LIN {X 0,Y 374.664,Z 501.893,A -85,B 0,C 180,E1 -12895.484,E2 -12895.484} C_VEL
LIN {X 0,Y 375.928,Z 486.688,A -85,B 0,C 180,E1 -12896.337,E2 -12896.337} C_VEL
LIN {X 0,Y 376.934,Z 471.292,A -85,B 0,C 180,E1 -12896.955,E2 -12896.955} C_VEL
LIN {X 0,Y 377.639,Z 455.754,A -85,B 0,C 180,E1 -12897.35,E2 -12897.35} C_VEL
LIN {X 0,Y 380.551,Z 335.489,A -85,B 0,C 180,E1 -12899.654,E2 -12899.654} C_VEL
LIN {X 0,Y 372.146,Z 316.425,A -85,B 0,C 180,E1 -12900.818,E2 -12900.818} C_VEL
LIN {X 0,Y 363.395,Z 298.754,A -85,B 0,C 180,E1 -12902.069,E2 -12902.069} C_VEL
LIN {X 0,Y 361.869,Z 293.041,A -85,B 0,C 180,E1 -12903.644,E2 -12903.644} C_VEL
LIN {X 0,Y 361.861,Z 293.034,A -85,B 0,C 180,E1 -12907.222,E2 -12907.222} C_VEL
LIN {X 0,Y 361.831,Z 293.031,A -85,B 0,C 180,E1 -12910.754,E2 -12910.754} C_VEL
LIN {X 0,Y 361.812,Z 293.041,A -85,B 0,C 180,E1 -12914.368,E2 -12914.368} C_VEL
LIN {X 0,Y 361.83,Z 293.025,A -85,B 0,C 180,E1 -12917.567,E2 -12917.567} C_VEL
LIN {X 0,Y 361.86,Z 293.038,A -85,B 0,C 180,E1 -12920.973,E2 -12920.973} C_VEL
LIN {X 0,Y 361.863,Z 293.025,A -85,B 0,C 180,E1 -12924.655,E2 -12924.655} C_VEL
LIN {X 0,Y 361.83,Z 293.023,A -85,B 0,C 180,E1 -12928.37,E2 -12928.37} C_VEL
LIN {X 0,Y 361.879,Z 293.031,A -85,B 0,C 180,E1 -12932.218,E2 -12932.218} C_VEL
LIN {X 0,Y 361.898,Z 293.029,A -85,B 0,C 180,E1 -12935.932,E2 -12935.932} C_VEL
LIN {X 0,Y 361.874,Z 293.033,A -85,B 0,C 180,E1 -12939.538,E2 -12939.538} C_VEL
LIN {X 0,Y 361.919,Z 293.024,A -85,B 0,C 180,E1 -12943.065,E2 -12943.065} C_VEL
LIN {X 0,Y 361.989,Z 293.013,A -85,B 0,C 180,E1 -12946.527,E2 -12946.527} C_VEL
LIN {X 0,Y 361.989,Z 293.016,A -85,B 0,C 180,E1 -12949.937,E2 -12949.937} C_VEL
LIN {X 0,Y 362.131,Z 293.001,A -85,B 0,C 180,E1 -12953.313,E2 -12953.313} C_VEL
LIN {X 0,Y 362.26,Z 292.984,A -85,B 0,C 180,E1 -12957.776,E2 -12957.776} C_VEL
LIN {X 0,Y 362.37,Z 292.964,A -85,B 0,C 180,E1 -12960,E2 -12960} C_VEL
LIN {X 0,Y 362.254,Z 292.985,A -85,B 0,C 180,E1 -12962.224,E2 -12962.224} C_VEL
LIN {X 0,Y 362.129,Z 293.005,A -85,B 0,C 180,E1 -12966.687,E2 -12966.687} C_VEL
LIN {X 0,Y 361.986,Z 293.014,A -85,B 0,C 180,E1 -12970.063,E2 -12970.063} C_VEL
LIN {X 0,Y 361.988,Z 293.011,A -85,B 0,C 180,E1 -12973.899,E2 -12973.899} C_VEL
LIN {X 0,Y 361.917,Z 293.024,A -85,B 0,C 180,E1 -12976.935,E2 -12976.935} C_VEL
LIN {X 0,Y 361.874,Z 293.035,A -85,B 0,C 180,E1 -12980.462,E2 -12980.462} C_VEL
LIN {X 0,Y 361.852,Z 293.04,A -85,B 0,C 180,E1 -12984.102,E2 -12984.102} C_VEL
LIN {X 0,Y 361.834,Z 293.039,A -85,B 0,C 180,E1 -12987.785,E2 -12987.785} C_VEL
LIN {X 0,Y 361.839,Z 293.037,A -85,B 0,C 180,E1 -12991.286,E2 -12991.286} C_VEL
LIN {X 0,Y 361.842,Z 293.037,A -85,B 0,C 180,E1 -12994.282,E2 -12994.282} C_VEL
LIN {X 0,Y 361.849,Z 293.034,A -85,B 0,C 180,E1 -12997.222,E2 -12997.222} C_VEL
LIN {X 0,Y 361.805,Z 293.021,A -85,B 0,C 180,E1 -13000.752,E2 -13000.752} C_VEL
LIN {X 0,Y 361.807,Z 293.04,A -85,B 0,C 180,E1 -13004.37,E2 -13004.37} C_VEL
LIN {X 0,Y 361.816,Z 293.042,A -85,B 0,C 180,E1 -13007.571,E2 -13007.571} C_VEL
LIN {X 0,Y 361.837,Z 293.035,A -85,B 0,C 180,E1 -13011.573,E2 -13011.573} C_VEL
LIN {X 0,Y 361.874,Z 293.078,A -85,B 0,C 180,E1 -13012.878,E2 -13012.878} C_VEL
LIN {X 0,Y 365.461,Z 306.162,A -85,B 0,C 180,E1 -13016.105,E2 -13016.105} C_VEL
LIN {X 0,Y 367.967,Z 316.314,A -85,B 0,C 180,E1 -13018.431,E2 -13018.431} C_VEL
LIN {X 0,Y 375.127,Z 332.742,A -85,B 0,C 180,E1 -13019.453,E2 -13019.453} C_VEL
LIN {X 0,Y 380.024,Z 358.744,A -85,B 0,C 180,E1 -13020.439,E2 -13020.439} C_VEL
LIN {X 0,Y 377.691,Z 458.455,A -85,B 0,C 180,E1 -13022.353,E2 -13022.353} C_VEL
LIN {X 0,Y 376.872,Z 484.598,A -85,B 0,C 180,E1 -13022.89,E2 -13022.89} C_VEL
LIN {X 0,Y 375.857,Z 500.037,A -85,B 0,C 180,E1 -13023.411,E2 -13023.411} C_VEL
LIN {X 0,Y 374.562,Z 514.958,A -85,B 0,C 180,E1 -13024.137,E2 -13024.137} C_VEL
LIN {X 0,Y 373.104,Z 528.815,A -85,B 0,C 180,E1 -13025.025,E2 -13025.025} C_VEL
LIN {X 0,Y 371.347,Z 542.584,A -85,B 0,C 180,E1 -13026.139,E2 -13026.139} C_VEL
LIN {X 0,Y 369.455,Z 556.024,A -85,B 0,C 180,E1 -13027.492,E2 -13027.492} C_VEL
LIN {X 0,Y 367.597,Z 568.269,A -85,B 0,C 180,E1 -13028.994,E2 -13028.994} C_VEL
LIN {X 0,Y 365.948,Z 579.825,A -85,B 0,C 180,E1 -13030.719,E2 -13030.719} C_VEL
LIN {X 0,Y 364.213,Z 590.313,A -85,B 0,C 180,E1 -13032.597,E2 -13032.597} C_VEL
LIN {X 0,Y 362.902,Z 599.362,A -85,B 0,C 180,E1 -13034.557,E2 -13034.557} C_VEL
LIN {X 0,Y 361.936,Z 606.874,A -85,B 0,C 180,E1 -13036.526,E2 -13036.526} C_VEL
LIN {X 0,Y 361.142,Z 613.884,A -85,B 0,C 180,E1 -13038.779,E2 -13038.779} C_VEL
LIN {X 0,Y 360.644,Z 619.4,A -85,B 0,C 180,E1 -13041.031,E2 -13041.031} C_VEL
LIN {X 0,Y 360.386,Z 623.572,A -85,B 0,C 180,E1 -13043.281,E2 -13043.281} C_VEL
LIN {X 0,Y 360.309,Z 626.5,A -85,B 0,C 180,E1 -13045.525,E2 -13045.525} C_VEL
LIN {X 0,Y 360.256,Z 628.244,A -85,B 0,C 180,E1 -13047.764,E2 -13047.764} C_VEL
LIN {X 0,Y 360.357,Z 628.844,A -85,B 0,C 180,E1 -13050,E2 -13050} C_VEL
LIN {X 0,Y 360.256,Z 628.237,A -85,B 0,C 180,E1 -13052.236,E2 -13052.236} C_VEL
LIN {X 0,Y 360.303,Z 626.484,A -85,B 0,C 180,E1 -13054.475,E2 -13054.475} C_VEL
LIN {X 0,Y 360.385,Z 623.553,A -85,B 0,C 180,E1 -13056.719,E2 -13056.719} C_VEL
LIN {X 0,Y 360.633,Z 619.38,A -85,B 0,C 180,E1 -13058.969,E2 -13058.969} C_VEL
LIN {X 0,Y 361.141,Z 613.854,A -85,B 0,C 180,E1 -13061.221,E2 -13061.221} C_VEL
LIN {X 0,Y 361.912,Z 606.826,A -85,B 0,C 180,E1 -13063.475,E2 -13063.475} C_VEL
LIN {X 0,Y 363.101,Z 598.089,A -85,B 0,C 180,E1 -13065.722,E2 -13065.722} C_VEL
LIN {X 0,Y 364.432,Z 588.811,A -85,B 0,C 180,E1 -13067.682,E2 -13067.682} C_VEL
LIN {X 0,Y 365.958,Z 579.723,A -85,B 0,C 180,E1 -13069.287,E2 -13069.287} C_VEL
LIN {X 0,Y 367.626,Z 568.19,A -85,B 0,C 180,E1 -13071.004,E2 -13071.004} C_VEL
LIN {X 0,Y 369.477,Z 555.931,A -85,B 0,C 180,E1 -13072.507,E2 -13072.507} C_VEL
LIN {X 0,Y 371.354,Z 542.454,A -85,B 0,C 180,E1 -13073.861,E2 -13073.861} C_VEL
LIN {X 0,Y 373.094,Z 528.68,A -85,B 0,C 180,E1 -13074.973,E2 -13074.973} C_VEL
LIN {X 0,Y 374.602,Z 514.187,A -85,B 0,C 180,E1 -13075.898,E2 -13075.898} C_VEL
LIN {X 0,Y 375.971,Z 498.225,A -85,B 0,C 180,E1 -13076.655,E2 -13076.655} C_VEL
LIN {X 0,Y 376.879,Z 483.026,A -85,B 0,C 180,E1 -13077.147,E2 -13077.147} C_VEL
LIN {X 0,Y 379.232,Z 393.182,A -85,B 0,C 180,E1 -13078.883,E2 -13078.883} C_VEL
LIN {X 0,Y 379.96,Z 358.776,A -85,B 0,C 180,E1 -13079.551,E2 -13079.551} C_VEL
LIN {X 0,Y 374.924,Z 332.033,A -85,B 0,C 180,E1 -13080.564,E2 -13080.564} C_VEL
LIN {X 0,Y 367.914,Z 315.979,A -85,B 0,C 180,E1 -13081.585,E2 -13081.585} C_VEL
LIN {X 0,Y 364.205,Z 301.343,A -85,B 0,C 180,E1 -13085.034,E2 -13085.034} C_VEL
LIN {X 0,Y 361.866,Z 293.036,A -85,B 0,C 180,E1 -13087.123,E2 -13087.123} C_VEL
LIN {X 0,Y 361.806,Z 293.044,A -85,B 0,C 180,E1 -13090.75,E2 -13090.75} C_VEL
LIN {X 0,Y 361.808,Z 293.044,A -85,B 0,C 180,E1 -13094.368,E2 -13094.368} C_VEL
LIN {X 0,Y 361.823,Z 293.039,A -85,B 0,C 180,E1 -13097.569,E2 -13097.569} C_VEL
LIN {X 0,Y 361.834,Z 293.037,A -85,B 0,C 180,E1 -13101.571,E2 -13101.571} C_VEL
LIN {X 0,Y 361.861,Z 293.031,A -85,B 0,C 180,E1 -13104.656,E2 -13104.656} C_VEL
LIN {X 0,Y 361.829,Z 293.038,A -85,B 0,C 180,E1 -13108.37,E2 -13108.37} C_VEL
LIN {X 0,Y 361.857,Z 293.033,A -85,B 0,C 180,E1 -13110.952,E2 -13110.952} C_VEL
LIN {X 0,Y 361.851,Z 293.035,A -85,B 0,C 180,E1 -13114.704,E2 -13114.704} C_VEL
LIN {X 0,Y 361.85,Z 293.033,A -85,B 0,C 180,E1 -13118.345,E2 -13118.345} C_VEL
LIN {X 0,Y 361.91,Z 293.011,A -85,B 0,C 180,E1 -13122.085,E2 -13122.085} C_VEL
LIN {X 0,Y 361.951,Z 293.024,A -85,B 0,C 180,E1 -13125.379,E2 -13125.379} C_VEL
LIN {X 0,Y 361.95,Z 292.993,A -85,B 0,C 180,E1 -13128.804,E2 -13128.804} C_VEL
LIN {X 0,Y 362.068,Z 293.008,A -85,B 0,C 180,E1 -13132.191,E2 -13132.191} C_VEL
LIN {X 0,Y 362.087,Z 292.997,A -85,B 0,C 180,E1 -13134.431,E2 -13134.431} C_VEL
LIN {X 0,Y 362.253,Z 292.98,A -85,B 0,C 180,E1 -13137.776,E2 -13137.776} C_VEL
LIN {X 0,Y 362.258,Z 292.978,A -85,B 0,C 180,E1 -13142.224,E2 -13142.224} C_VEL
LIN {X 0,Y 362.13,Z 292.996,A -85,B 0,C 180,E1 -13146.687,E2 -13146.687} C_VEL
LIN {X 0,Y 361.988,Z 293.014,A -85,B 0,C 180,E1 -13150.063,E2 -13150.063} C_VEL
LIN {X 0,Y 361.988,Z 293.015,A -85,B 0,C 180,E1 -13153.899,E2 -13153.899} C_VEL
LIN {X 0,Y 361.918,Z 293.029,A -85,B 0,C 180,E1 -13156.935,E2 -13156.935} C_VEL
LIN {X 0,Y 361.874,Z 293.008,A -85,B 0,C 180,E1 -13160.462,E2 -13160.462} C_VEL
LIN {X 0,Y 361.885,Z 293.03,A -85,B 0,C 180,E1 -13164.113,E2 -13164.113} C_VEL
LIN {X 0,Y 361.88,Z 293.013,A -85,B 0,C 180,E1 -13167.782,E2 -13167.782} C_VEL
LIN {X 0,Y 361.839,Z 293.035,A -85,B 0,C 180,E1 -13171.286,E2 -13171.286} C_VEL
LIN {X 0,Y 361.843,Z 293.036,A -85,B 0,C 180,E1 -13174.282,E2 -13174.282} C_VEL
LIN {X 0,Y 361.854,Z 293.032,A -85,B 0,C 180,E1 -13177.223,E2 -13177.223} C_VEL
LIN {X 0,Y 361.829,Z 293.037,A -85,B 0,C 180,E1 -13180.756,E2 -13180.756} C_VEL
LIN {X 0,Y 361.812,Z 293.041,A -85,B 0,C 180,E1 -13184.369,E2 -13184.369} C_VEL
LIN {X 0,Y 361.832,Z 293.039,A -85,B 0,C 180,E1 -13187.569,E2 -13187.569} C_VEL
LIN {X 0,Y 361.866,Z 293.026,A -85,B 0,C 180,E1 -13190.974,E2 -13190.974} C_VEL
LIN {X 0,Y 361.871,Z 293.028,A -85,B 0,C 180,E1 -13194.656,E2 -13194.656} C_VEL
LIN {X 0,Y 361.871,Z 293.2,A -85,B 0,C 180,E1 -13196.547,E2 -13196.547} C_VEL
LIN {X 0,Y 363.492,Z 299.001,A -85,B 0,C 180,E1 -13198.071,E2 -13198.071} C_VEL
LIN {X 0,Y 374.141,Z 320.751,A -85,B 0,C 180,E1 -13199.567,E2 -13199.567} C_VEL
LIN {X 0,Y 380.491,Z 335.431,A -85,B 0,C 180,E1 -13200.445,E2 -13200.445} C_VEL
LIN {X 0,Y 378.084,Z 434.705,A -85,B 0,C 180,E1 -13202.347,E2 -13202.347} C_VEL
LIN {X 0,Y 377.196,Z 464.75,A -85,B 0,C 180,E1 -13202.952,E2 -13202.952} C_VEL
LIN {X 0,Y 376.39,Z 480.281,A -85,B 0,C 180,E1 -13203.484,E2 -13203.484} C_VEL
LIN {X 0,Y 375.345,Z 494.194,A -85,B 0,C 180,E1 -13204.156,E2 -13204.156} C_VEL
LIN {X 0,Y 374.115,Z 507.436,A -85,B 0,C 180,E1 -13204.997,E2 -13204.997} C_VEL
LIN {X 0,Y 372.454,Z 521.009,A -85,B 0,C 180,E1 -13206.066,E2 -13206.066} C_VEL
LIN {X 0,Y 370.69,Z 534.773,A -85,B 0,C 180,E1 -13207.424,E2 -13207.424} C_VEL
LIN {X 0,Y 368.995,Z 546.126,A -85,B 0,C 180,E1 -13208.785,E2 -13208.785} C_VEL
LIN {X 0,Y 367.249,Z 557.582,A -85,B 0,C 180,E1 -13210.434,E2 -13210.434} C_VEL
LIN {X 0,Y 365.692,Z 567.22,A -85,B 0,C 180,E1 -13212.092,E2 -13212.092} C_VEL
LIN {X 0,Y 364.187,Z 576.663,A -85,B 0,C 180,E1 -13214.039,E2 -13214.039} C_VEL
LIN {X 0,Y 363.002,Z 584.521,A -85,B 0,C 180,E1 -13215.995,E2 -13215.995} C_VEL
LIN {X 0,Y 362.214,Z 590.183,A -85,B 0,C 180,E1 -13217.677,E2 -13217.677} C_VEL
LIN {X 0,Y 361.42,Z 596.35,A -85,B 0,C 180,E1 -13219.921,E2 -13219.921} C_VEL
LIN {X 0,Y 360.905,Z 601.111,A -85,B 0,C 180,E1 -13222.166,E2 -13222.166} C_VEL
LIN {X 0,Y 360.586,Z 604.598,A -85,B 0,C 180,E1 -13224.408,E2 -13224.408} C_VEL
LIN {X 0,Y 360.374,Z 606.904,A -85,B 0,C 180,E1 -13226.646,E2 -13226.646} C_VEL
LIN {X 0,Y 360.348,Z 608.08,A -85,B 0,C 180,E1 -13228.883,E2 -13228.883} C_VEL
LIN {X 0,Y 360.348,Z 608.095,A -85,B 0,C 180,E1 -13231.118,E2 -13231.118} C_VEL
LIN {X 0,Y 360.369,Z 606.98,A -85,B 0,C 180,E1 -13233.354,E2 -13233.354} C_VEL
LIN {X 0,Y 360.57,Z 604.732,A -85,B 0,C 180,E1 -13235.593,E2 -13235.593} C_VEL
LIN {X 0,Y 360.872,Z 601.3,A -85,B 0,C 180,E1 -13237.835,E2 -13237.835} C_VEL
LIN {X 0,Y 361.385,Z 596.6,A -85,B 0,C 180,E1 -13240.08,E2 -13240.08} C_VEL
LIN {X 0,Y 362.244,Z 590.194,A -85,B 0,C 180,E1 -13242.421,E2 -13242.421} C_VEL
LIN {X 0,Y 363.065,Z 583.887,A -85,B 0,C 180,E1 -13244.288,E2 -13244.288} C_VEL
LIN {X 0,Y 364.319,Z 575.879,A -85,B 0,C 180,E1 -13246.243,E2 -13246.243} C_VEL
LIN {X 0,Y 364.568,Z 574.52,A -85,B 0,C 180,E1 -13246.547,E2 -13246.547} C_VEL
LIN {X 0,Y 364.5,Z 571.102,A -85,B 0,C 180,E1 -13247.293,E2 -13247.293} C_VEL
LIN {X 0,Y 362.703,Z 565.43,A -85,B 0,C 180,E1 -13248.538,E2 -13248.538} C_VEL
LIN {X 0,Y 360.981,Z 559.353,A -85,B 0,C 180,E1 -13249.758,E2 -13249.758} C_VEL
LIN {X 0,Y 361.007,Z 555.28,A -85,B 0,C 180,E1 -13250.443,E2 -13250.443} C_VEL
LIN {X 0,Y 362.764,Z 543.878,A -85,B 0,C 180,E1 -13252.046,E2 -13252.046} C_VEL
LIN {X 0,Y 364.597,Z 532.01,A -85,B 0,C 180,E1 -13253.426,E2 -13253.426} C_VEL
LIN {X 0,Y 366.32,Z 519.162,A -85,B 0,C 180,E1 -13254.662,E2 -13254.662} C_VEL
LIN {X 0,Y 367.952,Z 505.063,A -85,B 0,C 180,E1 -13255.755,E2 -13255.755} C_VEL
LIN {X 0,Y 369.36,Z 489.844,A -85,B 0,C 180,E1 -13256.669,E2 -13256.669} C_VEL
LIN {X 0,Y 370.399,Z 475.161,A -85,B 0,C 180,E1 -13257.318,E2 -13257.318} C_VEL
LIN {X 0,Y 371.184,Z 460.482,A -85,B 0,C 180,E1 -13257.752,E2 -13257.752} C_VEL
LIN {X 0,Y 374.403,Z 337.801,A -85,B 0,C 180,E1 -13260.144,E2 -13260.144} C_VEL
LIN {X 0,Y 368.077,Z 323.029,A -85,B 0,C 180,E1 -13261.052,E2 -13261.052} C_VEL
LIN {X 0,Y 359.045,Z 304.685,A -85,B 0,C 180,E1 -13262.355,E2 -13262.355} C_VEL
LIN {X 0,Y 356.106,Z 298.924,A -85,B 0,C 180,E1 -13262.823,E2 -13262.823} C_VEL
LIN {X 0,Y 354.807,Z 293.915,A -85,B 0,C 180,E1 -13264.239,E2 -13264.239} C_VEL
LIN {X 0,Y 354.803,Z 293.915,A -85,B 0,C 180,E1 -13267.882,E2 -13267.882} C_VEL
LIN {X 0,Y 354.784,Z 293.912,A -85,B 0,C 180,E1 -13271.171,E2 -13271.171} C_VEL
LIN {X 0,Y 354.758,Z 293.92,A -85,B 0,C 180,E1 -13274.505,E2 -13274.505} C_VEL
LIN {X 0,Y 354.788,Z 293.901,A -85,B 0,C 180,E1 -13277.662,E2 -13277.662} C_VEL
LIN {X 0,Y 354.81,Z 293.913,A -85,B 0,C 180,E1 -13280.665,E2 -13280.665} C_VEL
LIN {X 0,Y 354.812,Z 293.901,A -85,B 0,C 180,E1 -13284.301,E2 -13284.301} C_VEL
LIN {X 0,Y 354.779,Z 293.908,A -85,B 0,C 180,E1 -13287.666,E2 -13287.666} C_VEL
LIN {X 0,Y 354.813,Z 293.912,A -85,B 0,C 180,E1 -13291.616,E2 -13291.616} C_VEL
LIN {X 0,Y 354.866,Z 293.901,A -85,B 0,C 180,E1 -13294.17,E2 -13294.17} C_VEL
LIN {X 0,Y 354.799,Z 293.908,A -85,B 0,C 180,E1 -13297.892,E2 -13297.892} C_VEL
LIN {X 0,Y 354.842,Z 293.903,A -85,B 0,C 180,E1 -13301.525,E2 -13301.525} C_VEL
LIN {X 0,Y 354.909,Z 293.899,A -85,B 0,C 180,E1 -13305.082,E2 -13305.082} C_VEL
LIN {X 0,Y 354.922,Z 293.9,A -85,B 0,C 180,E1 -13308.579,E2 -13308.579} C_VEL
LIN {X 0,Y 355.052,Z 293.878,A -85,B 0,C 180,E1 -13312.035,E2 -13312.035} C_VEL
LIN {X 0,Y 355.066,Z 293.882,A -85,B 0,C 180,E1 -13314.32,E2 -13314.32} C_VEL
LIN {X 0,Y 355.222,Z 293.86,A -85,B 0,C 180,E1 -13317.732,E2 -13317.732} C_VEL
LIN {X 0,Y 355.321,Z 293.841,A -85,B 0,C 180,E1 -13320,E2 -13320} C_VEL
LIN {X 0,Y 355.217,Z 293.862,A -85,B 0,C 180,E1 -13322.268,E2 -13322.268} C_VEL
LIN {X 0,Y 355.094,Z 293.88,A -85,B 0,C 180,E1 -13326.82,E2 -13326.82} C_VEL
LIN {X 0,Y 354.943,Z 293.893,A -85,B 0,C 180,E1 -13330.265,E2 -13330.265} C_VEL
LIN {X 0,Y 354.933,Z 293.891,A -85,B 0,C 180,E1 -13334.018,E2 -13334.018} C_VEL
LIN {X 0,Y 354.88,Z 293.899,A -85,B 0,C 180,E1 -13338.092,E2 -13338.092} C_VEL
LIN {X 0,Y 354.797,Z 293.91,A -85,B 0,C 180,E1 -13342.108,E2 -13342.108} C_VEL
LIN {X 0,Y 354.797,Z 293.91,A -85,B 0,C 180,E1 -13345.835,E2 -13345.835} C_VEL
LIN {X 0,Y 354.788,Z 293.916,A -85,B 0,C 180,E1 -13349.684,E2 -13349.684} C_VEL
LIN {X 0,Y 354.778,Z 293.913,A -85,B 0,C 180,E1 -13352.334,E2 -13352.334} C_VEL
LIN {X 0,Y 354.81,Z 293.912,A -85,B 0,C 180,E1 -13355.699,E2 -13355.699} C_VEL
LIN {X 0,Y 354.761,Z 293.908,A -85,B 0,C 180,E1 -13359.413,E2 -13359.413} C_VEL
LIN {X 0,Y 354.778,Z 293.917,A -85,B 0,C 180,E1 -13362.867,E2 -13362.867} C_VEL
LIN {X 0,Y 354.756,Z 293.918,A -85,B 0,C 180,E1 -13366.103,E2 -13366.103} C_VEL
LIN {X 0,Y 354.757,Z 293.919,A -85,B 0,C 180,E1 -13369.176,E2 -13369.176} C_VEL
LIN {X 0,Y 354.813,Z 293.951,A -85,B 0,C 180,E1 -13372.264,E2 -13372.264} C_VEL
LIN {X 0,Y 358.306,Z 306.545,A -85,B 0,C 180,E1 -13375.468,E2 -13375.468} C_VEL
LIN {X 0,Y 360.733,Z 316.15,A -85,B 0,C 180,E1 -13377.723,E2 -13377.723} C_VEL
LIN {X 0,Y 369.28,Z 335.281,A -85,B 0,C 180,E1 -13378.977,E2 -13378.977} C_VEL
LIN {X 0,Y 373.846,Z 359.885,A -85,B 0,C 180,E1 -13379.929,E2 -13379.929} C_VEL
LIN {X 0,Y 371.263,Z 463.643,A -85,B 0,C 180,E1 -13381.948,E2 -13381.948} C_VEL
LIN {X 0,Y 370.496,Z 485.548,A -85,B 0,C 180,E1 -13382.422,E2 -13382.422} C_VEL
LIN {X 0,Y 369.448,Z 500.604,A -85,B 0,C 180,E1 -13382.951,E2 -13382.951} C_VEL
LIN {X 0,Y 368.171,Z 514.752,A -85,B 0,C 180,E1 -13383.653,E2 -13383.653} C_VEL
LIN {X 0,Y 366.603,Z 529.004,A -85,B 0,C 180,E1 -13384.584,E2 -13384.584} C_VEL
LIN {X 0,Y 364.852,Z 542.384,A -85,B 0,C 180,E1 -13385.687,E2 -13385.687} C_VEL
LIN {X 0,Y 362.876,Z 555.824,A -85,B 0,C 180,E1 -13387.06,E2 -13387.06} C_VEL
LIN {X 0,Y 360.915,Z 568.067,A -85,B 0,C 180,E1 -13388.586,E2 -13388.586} C_VEL
LIN {X 0,Y 359.149,Z 579.797,A -85,B 0,C 180,E1 -13390.371,E2 -13390.371} C_VEL
LIN {X 0,Y 357.359,Z 590.11,A -85,B 0,C 180,E1 -13392.253,E2 -13392.253} C_VEL
LIN {X 0,Y 355.992,Z 599.159,A -85,B 0,C 180,E1 -13394.25,E2 -13394.25} C_VEL
LIN {X 0,Y 354.938,Z 606.669,A -85,B 0,C 180,E1 -13396.255,E2 -13396.255} C_VEL
LIN {X 0,Y 354.137,Z 613.681,A -85,B 0,C 180,E1 -13398.554,E2 -13398.554} C_VEL
LIN {X 0,Y 353.585,Z 619.196,A -85,B 0,C 180,E1 -13400.851,E2 -13400.851} C_VEL
LIN {X 0,Y 353.305,Z 623.369,A -85,B 0,C 180,E1 -13403.145,E2 -13403.145} C_VEL
LIN {X 0,Y 353.224,Z 626.297,A -85,B 0,C 180,E1 -13405.435,E2 -13405.435} C_VEL
LIN {X 0,Y 353.164,Z 628.041,A -85,B 0,C 180,E1 -13407.719,E2 -13407.719} C_VEL
LIN {X 0,Y 353.26,Z 628.641,A -85,B 0,C 180,E1 -13410,E2 -13410} C_VEL
LIN {X 0,Y 353.164,Z 628.034,A -85,B 0,C 180,E1 -13412.281,E2 -13412.281} C_VEL
LIN {X 0,Y 353.218,Z 626.28,A -85,B 0,C 180,E1 -13414.565,E2 -13414.565} C_VEL
LIN {X 0,Y 353.302,Z 623.349,A -85,B 0,C 180,E1 -13416.855,E2 -13416.855} C_VEL
LIN {X 0,Y 353.578,Z 619.175,A -85,B 0,C 180,E1 -13419.149,E2 -13419.149} C_VEL
LIN {X 0,Y 354.137,Z 613.649,A -85,B 0,C 180,E1 -13421.446,E2 -13421.446} C_VEL
LIN {X 0,Y 354.892,Z 606.618,A -85,B 0,C 180,E1 -13423.747,E2 -13423.747} C_VEL
LIN {X 0,Y 356.194,Z 597.882,A -85,B 0,C 180,E1 -13426.035,E2 -13426.035} C_VEL
LIN {X 0,Y 357.627,Z 588.604,A -85,B 0,C 180,E1 -13428.029,E2 -13428.029} C_VEL
LIN {X 0,Y 359.333,Z 578.477,A -85,B 0,C 180,E1 -13429.837,E2 -13429.837} C_VEL
LIN {X 0,Y 361.075,Z 566.956,A -85,B 0,C 180,E1 -13431.554,E2 -13431.554} C_VEL
LIN {X 0,Y 363.08,Z 554.5,A -85,B 0,C 180,E1 -13433.076,E2 -13433.076} C_VEL
LIN {X 0,Y 364.852,Z 542.247,A -85,B 0,C 180,E1 -13434.313,E2 -13434.313} C_VEL
LIN {X 0,Y 366.763,Z 527.527,A -85,B 0,C 180,E1 -13435.513,E2 -13435.513} C_VEL
LIN {X 0,Y 368.269,Z 513.406,A -85,B 0,C 180,E1 -13436.416,E2 -13436.416} C_VEL
LIN {X 0,Y 369.65,Z 498.013,A -85,B 0,C 180,E1 -13437.148,E2 -13437.148} C_VEL
LIN {X 0,Y 370.591,Z 482.809,A -85,B 0,C 180,E1 -13437.647,E2 -13437.647} C_VEL
LIN {X 0,Y 373.227,Z 384.941,A -85,B 0,C 180,E1 -13439.566,E2 -13439.566} C_VEL
LIN {X 0,Y 373.78,Z 359.899,A -85,B 0,C 180,E1 -13440.06,E2 -13440.06} C_VEL
LIN {X 0,Y 368.962,Z 334.334,A -85,B 0,C 180,E1 -13441.056,E2 -13441.056} C_VEL
LIN {X 0,Y 360.631,Z 315.761,A -85,B 0,C 180,E1 -13442.295,E2 -13442.295} C_VEL
LIN {X 0,Y 357.381,Z 302.947,A -85,B 0,C 180,E1 -13445.399,E2 -13445.399} C_VEL
LIN {X 0,Y 354.793,Z 293.917,A -85,B 0,C 180,E1 -13447.739,E2 -13447.739} C_VEL
LIN {X 0,Y 354.765,Z 293.92,A -85,B 0,C 180,E1 -13451.167,E2 -13451.167} C_VEL
LIN {X 0,Y 354.755,Z 293.922,A -85,B 0,C 180,E1 -13454.505,E2 -13454.505} C_VEL
LIN {X 0,Y 354.781,Z 293.916,A -85,B 0,C 180,E1 -13457.661,E2 -13457.661} C_VEL
LIN {X 0,Y 354.778,Z 293.917,A -85,B 0,C 180,E1 -13460.661,E2 -13460.661} C_VEL
LIN {X 0,Y 354.81,Z 293.909,A -85,B 0,C 180,E1 -13464.301,E2 -13464.301} C_VEL
LIN {X 0,Y 354.778,Z 293.914,A -85,B 0,C 180,E1 -13467.666,E2 -13467.666} C_VEL
LIN {X 0,Y 354.79,Z 293.918,A -85,B 0,C 180,E1 -13471.614,E2 -13471.614} C_VEL
LIN {X 0,Y 354.795,Z 293.915,A -85,B 0,C 180,E1 -13475.419,E2 -13475.419} C_VEL
LIN {X 0,Y 354.815,Z 293.907,A -85,B 0,C 180,E1 -13479.113,E2 -13479.113} C_VEL
LIN {X 0,Y 354.87,Z 293.896,A -85,B 0,C 180,E1 -13482.719,E2 -13482.719} C_VEL
LIN {X 0,Y 354.941,Z 293.889,A -85,B 0,C 180,E1 -13486.255,E2 -13486.255} C_VEL
LIN {X 0,Y 354.938,Z 293.875,A -85,B 0,C 180,E1 -13489.735,E2 -13489.735} C_VEL
LIN {X 0,Y 355.087,Z 293.88,A -85,B 0,C 180,E1 -13493.18,E2 -13493.18} C_VEL
LIN {X 0,Y 355.216,Z 293.857,A -85,B 0,C 180,E1 -13497.732,E2 -13497.732} C_VEL
LIN {X 0,Y 355.22,Z 293.855,A -85,B 0,C 180,E1 -13502.268,E2 -13502.268} C_VEL
LIN {X 0,Y 355.095,Z 293.872,A -85,B 0,C 180,E1 -13506.82,E2 -13506.82} C_VEL
LIN {X 0,Y 354.945,Z 293.892,A -85,B 0,C 180,E1 -13510.265,E2 -13510.265} C_VEL
LIN {X 0,Y 354.933,Z 293.894,A -85,B 0,C 180,E1 -13514.019,E2 -13514.019} C_VEL
LIN {X 0,Y 354.881,Z 293.9,A -85,B 0,C 180,E1 -13518.093,E2 -13518.093} C_VEL
LIN {X 0,Y 354.808,Z 293.903,A -85,B 0,C 180,E1 -13522.108,E2 -13522.108} C_VEL
LIN {X 0,Y 354.866,Z 293.897,A -85,B 0,C 180,E1 -13525.83,E2 -13525.83} C_VEL
LIN {X 0,Y 354.81,Z 293.912,A -85,B 0,C 180,E1 -13529.683,E2 -13529.683} C_VEL
LIN {X 0,Y 354.8,Z 293.913,A -85,B 0,C 180,E1 -13533.703,E2 -13533.703} C_VEL
LIN {X 0,Y 354.788,Z 293.916,A -85,B 0,C 180,E1 -13536.461,E2 -13536.461} C_VEL
LIN {X 0,Y 354.819,Z 293.909,A -85,B 0,C 180,E1 -13539.425,E2 -13539.425} C_VEL
LIN {X 0,Y 354.783,Z 293.915,A -85,B 0,C 180,E1 -13542.868,E2 -13542.868} C_VEL
LIN {X 0,Y 354.762,Z 293.92,A -85,B 0,C 180,E1 -13546.104,E2 -13546.104} C_VEL
LIN {X 0,Y 354.784,Z 293.919,A -85,B 0,C 180,E1 -13549.18,E2 -13549.18} C_VEL
LIN {X 0,Y 354.804,Z 293.913,A -85,B 0,C 180,E1 -13552.403,E2 -13552.403} C_VEL
LIN {X 0,Y 354.817,Z 294.003,A -85,B 0,C 180,E1 -13555.934,E2 -13555.934} C_VEL
LIN {X 0,Y 356.242,Z 299.151,A -85,B 0,C 180,E1 -13557.338,E2 -13557.338} C_VEL
LIN {X 0,Y 367.052,Z 320.845,A -85,B 0,C 180,E1 -13558.911,E2 -13558.911} C_VEL
LIN {X 0,Y 374.267,Z 337.264,A -85,B 0,C 180,E1 -13559.938,E2 -13559.938} C_VEL
LIN {X 0,Y 372.146,Z 423.356,A -85,B 0,C 180,E1 -13561.618,E2 -13561.618} C_VEL
LIN {X 0,Y 370.97,Z 463.804,A -85,B 0,C 180,E1 -13562.422,E2 -13562.422} C_VEL
LIN {X 0,Y 370.128,Z 479.45,A -85,B 0,C 180,E1 -13562.948,E2 -13562.948} C_VEL
LIN {X 0,Y 369.003,Z 493.852,A -85,B 0,C 180,E1 -13563.644,E2 -13563.644} C_VEL
LIN {X 0,Y 367.702,Z 507.645,A -85,B 0,C 180,E1 -13564.53,E2 -13564.53} C_VEL
LIN {X 0,Y 365.958,Z 521.218,A -85,B 0,C 180,E1 -13565.614,E2 -13565.614} C_VEL
LIN {X 0,Y 364.136,Z 534.981,A -85,B 0,C 180,E1 -13566.994,E2 -13566.994} C_VEL
LIN {X 0,Y 362.374,Z 546.333,A -85,B 0,C 180,E1 -13568.378,E2 -13568.378} C_VEL
LIN {X 0,Y 360.565,Z 557.788,A -85,B 0,C 180,E1 -13570.056,E2 -13570.056} C_VEL
LIN {X 0,Y 358.928,Z 567.426,A -85,B 0,C 180,E1 -13571.743,E2 -13571.743} C_VEL
LIN {X 0,Y 357.342,Z 576.869,A -85,B 0,C 180,E1 -13573.725,E2 -13573.725} C_VEL
LIN {X 0,Y 356.057,Z 584.728,A -85,B 0,C 180,E1 -13575.716,E2 -13575.716} C_VEL
LIN {X 0,Y 355.27,Z 590.388,A -85,B 0,C 180,E1 -13577.432,E2 -13577.432} C_VEL
LIN {X 0,Y 354.399,Z 596.556,A -85,B 0,C 180,E1 -13579.719,E2 -13579.719} C_VEL
LIN {X 0,Y 353.854,Z 601.315,A -85,B 0,C 180,E1 -13582.009,E2 -13582.009} C_VEL
LIN {X 0,Y 353.509,Z 604.802,A -85,B 0,C 180,E1 -13584.295,E2 -13584.295} C_VEL
LIN {X 0,Y 353.296,Z 607.107,A -85,B 0,C 180,E1 -13586.579,E2 -13586.579} C_VEL
LIN {X 0,Y 353.25,Z 608.283,A -85,B 0,C 180,E1 -13588.86,E2 -13588.86} C_VEL
LIN {X 0,Y 353.25,Z 608.298,A -85,B 0,C 180,E1 -13591.14,E2 -13591.14} C_VEL
LIN {X 0,Y 353.291,Z 607.182,A -85,B 0,C 180,E1 -13593.421,E2 -13593.421} C_VEL
LIN {X 0,Y 353.49,Z 604.935,A -85,B 0,C 180,E1 -13595.705,E2 -13595.705} C_VEL
LIN {X 0,Y 353.807,Z 601.503,A -85,B 0,C 180,E1 -13597.993,E2 -13597.993} C_VEL
LIN {X 0,Y 354.352,Z 596.803,A -85,B 0,C 180,E1 -13600.282,E2 -13600.282} C_VEL
LIN {X 0,Y 355.246,Z 590.709,A -85,B 0,C 180,E1 -13602.569,E2 -13602.569} C_VEL
LIN {X 0,Y 356.163,Z 583.982,A -85,B 0,C 180,E1 -13604.603,E2 -13604.603} C_VEL
LIN {X 0,Y 357.707,Z 574.849,A -85,B 0,C 180,E1 -13606.845,E2 -13606.845} C_VEL
LIN {X 0,Y 359.383,Z 564.983,A -85,B 0,C 180,E1 -13608.824,E2 -13608.824} C_VEL
LIN {X 0,Y 361.007,Z 555.28,A -85,B 0,C 180,E1 -13610.443,E2 -13610.443} C_VEL
LIN {X 0,Y 361.08,Z 551.142,A -85,B 0,C 180,E1 -13611.11,E2 -13611.11} C_VEL
LIN {X 0,Y 359.546,Z 544.305,A -85,B 0,C 180,E1 -13612.223,E2 -13612.223} C_VEL
LIN {X 0,Y 358,Z 537.141,A -85,B 0,C 180,E1 -13613.282,E2 -13613.282} C_VEL
LIN {X 0,Y 358.041,Z 532.426,A -85,B 0,C 180,E1 -13613.855,E2 -13613.855} C_VEL
LIN {X 0,Y 359.888,Z 519.359,A -85,B 0,C 180,E1 -13615.133,E2 -13615.133} C_VEL
LIN {X 0,Y 361.585,Z 505.259,A -85,B 0,C 180,E1 -13616.242,E2 -13616.242} C_VEL
LIN {X 0,Y 363.025,Z 490.072,A -85,B 0,C 180,E1 -13617.17,E2 -13617.17} C_VEL
LIN {X 0,Y 364.105,Z 475.351,A -85,B 0,C 180,E1 -13617.83,E2 -13617.83} C_VEL
LIN {X 0,Y 364.935,Z 460.664,A -85,B 0,C 180,E1 -13618.269,E2 -13618.269} C_VEL
LIN {X 0,Y 368.241,Z 339.595,A -85,B 0,C 180,E1 -13620.667,E2 -13620.667} C_VEL
LIN {X 0,Y 360.756,Z 322.609,A -85,B 0,C 180,E1 -13621.769,E2 -13621.769} C_VEL
LIN {X 0,Y 352.578,Z 306.286,A -85,B 0,C 180,E1 -13622.989,E2 -13622.989} C_VEL
LIN {X 0,Y 348.976,Z 299.215,A -85,B 0,C 180,E1 -13623.567,E2 -13623.567} C_VEL
LIN {X 0,Y 347.764,Z 294.792,A -85,B 0,C 180,E1 -13624.856,E2 -13624.856} C_VEL
LIN {X 0,Y 347.749,Z 294.799,A -85,B 0,C 180,E1 -13628.792,E2 -13628.792} C_VEL
LIN {X 0,Y 347.747,Z 294.796,A -85,B 0,C 180,E1 -13631.829,E2 -13631.829} C_VEL
LIN {X 0,Y 347.701,Z 294.798,A -85,B 0,C 180,E1 -13635.026,E2 -13635.026} C_VEL
LIN {X 0,Y 347.744,Z 294.776,A -85,B 0,C 180,E1 -13638.397,E2 -13638.397} C_VEL
LIN {X 0,Y 347.765,Z 294.783,A -85,B 0,C 180,E1 -13642.011,E2 -13642.011} C_VEL
LIN {X 0,Y 347.736,Z 294.795,A -85,B 0,C 180,E1 -13645.535,E2 -13645.535} C_VEL
LIN {X 0,Y 347.737,Z 294.778,A -85,B 0,C 180,E1 -13648.299,E2 -13648.299} C_VEL
LIN {X 0,Y 347.753,Z 294.78,A -85,B 0,C 180,E1 -13650.985,E2 -13650.985} C_VEL
LIN {X 0,Y 347.803,Z 294.782,A -85,B 0,C 180,E1 -13653.605,E2 -13653.605} C_VEL
LIN {X 0,Y 347.773,Z 294.788,A -85,B 0,C 180,E1 -13656.161,E2 -13656.161} C_VEL
LIN {X 0,Y 347.795,Z 294.786,A -85,B 0,C 180,E1 -13659.908,E2 -13659.908} C_VEL
LIN {X 0,Y 347.822,Z 294.782,A -85,B 0,C 180,E1 -13663.568,E2 -13663.568} C_VEL
LIN {X 0,Y 347.879,Z 294.772,A -85,B 0,C 180,E1 -13667.16,E2 -13667.16} C_VEL
LIN {X 0,Y 347.925,Z 294.764,A -85,B 0,C 180,E1 -13670.7,E2 -13670.7} C_VEL
LIN {X 0,Y 348.062,Z 294.755,A -85,B 0,C 180,E1 -13673.041,E2 -13673.041} C_VEL
LIN {X 0,Y 348.184,Z 294.737,A -85,B 0,C 180,E1 -13677.686,E2 -13677.686} C_VEL
LIN {X 0,Y 348.272,Z 294.719,A -85,B 0,C 180,E1 -13680,E2 -13680} C_VEL
LIN {X 0,Y 348.179,Z 294.74,A -85,B 0,C 180,E1 -13682.314,E2 -13682.314} C_VEL
LIN {X 0,Y 348.061,Z 294.755,A -85,B 0,C 180,E1 -13686.958,E2 -13686.958} C_VEL
LIN {X 0,Y 347.883,Z 294.775,A -85,B 0,C 180,E1 -13690.476,E2 -13690.476} C_VEL
LIN {X 0,Y 347.89,Z 294.769,A -85,B 0,C 180,E1 -13694.15,E2 -13694.15} C_VEL
LIN {X 0,Y 347.82,Z 294.779,A -85,B 0,C 180,E1 -13698.259,E2 -13698.259} C_VEL
LIN {X 0,Y 347.754,Z 294.788,A -85,B 0,C 180,E1 -13701.625,E2 -13701.625} C_VEL
LIN {X 0,Y 347.731,Z 294.792,A -85,B 0,C 180,E1 -13705.115,E2 -13705.115} C_VEL
LIN {X 0,Y 347.728,Z 294.796,A -85,B 0,C 180,E1 -13707.701,E2 -13707.701} C_VEL
LIN {X 0,Y 347.73,Z 294.796,A -85,B 0,C 180,E1 -13710.35,E2 -13710.35} C_VEL
LIN {X 0,Y 347.74,Z 294.79,A -85,B 0,C 180,E1 -13714.044,E2 -13714.044} C_VEL
LIN {X 0,Y 347.746,Z 294.791,A -85,B 0,C 180,E1 -13717.323,E2 -13717.323} C_VEL
LIN {X 0,Y 347.69,Z 294.779,A -85,B 0,C 180,E1 -13720.303,E2 -13720.303} C_VEL
LIN {X 0,Y 347.716,Z 294.798,A -85,B 0,C 180,E1 -13723.409,E2 -13723.409} C_VEL
LIN {X 0,Y 347.716,Z 294.795,A -85,B 0,C 180,E1 -13726.688,E2 -13726.688} C_VEL
LIN {X 0,Y 347.695,Z 294.797,A -85,B 0,C 180,E1 -13730.183,E2 -13730.183} C_VEL
LIN {X 0,Y 347.732,Z 294.837,A -85,B 0,C 180,E1 -13731.619,E2 -13731.619} C_VEL
LIN {X 0,Y 351.156,Z 306.814,A -85,B 0,C 180,E1 -13734.774,E2 -13734.774} C_VEL
LIN {X 0,Y 353.405,Z 315.714,A -85,B 0,C 180,E1 -13736.965,E2 -13736.965} C_VEL
LIN {X 0,Y 362.444,Z 335.549,A -85,B 0,C 180,E1 -13738.335,E2 -13738.335} C_VEL
LIN {X 0,Y 363.675,Z 339.128,A -85,B 0,C 180,E1 -13738.535,E2 -13738.535} C_VEL
LIN {X 0,Y 367.691,Z 361.135,A -85,B 0,C 180,E1 -13739.404,E2 -13739.404} C_VEL
LIN {X 0,Y 364.974,Z 465.251,A -85,B 0,C 180,E1 -13741.46,E2 -13741.46} C_VEL
LIN {X 0,Y 364.211,Z 485.358,A -85,B 0,C 180,E1 -13741.905,E2 -13741.905} C_VEL
LIN {X 0,Y 363.149,Z 500.41,A -85,B 0,C 180,E1 -13742.442,E2 -13742.442} C_VEL
LIN {X 0,Y 361.809,Z 514.555,A -85,B 0,C 180,E1 -13743.153,E2 -13743.153} C_VEL
LIN {X 0,Y 360.267,Z 528.19,A -85,B 0,C 180,E1 -13744.051,E2 -13744.051} C_VEL
LIN {X 0,Y 358.376,Z 542.185,A -85,B 0,C 180,E1 -13745.218,E2 -13745.218} C_VEL
LIN {X 0,Y 356.314,Z 555.623,A -85,B 0,C 180,E1 -13746.613,E2 -13746.613} C_VEL
LIN {X 0,Y 354.23,Z 567.864,A -85,B 0,C 180,E1 -13748.161,E2 -13748.161} C_VEL
LIN {X 0,Y 352.464,Z 579.188,A -85,B 0,C 180,E1 -13749.907,E2 -13749.907} C_VEL
LIN {X 0,Y 350.552,Z 589.907,A -85,B 0,C 180,E1 -13751.896,E2 -13751.896} C_VEL
LIN {X 0,Y 349.104,Z 598.956,A -85,B 0,C 180,E1 -13753.931,E2 -13753.931} C_VEL
LIN {X 0,Y 347.955,Z 606.465,A -85,B 0,C 180,E1 -13755.974,E2 -13755.974} C_VEL
LIN {X 0,Y 347.108,Z 613.477,A -85,B 0,C 180,E1 -13758.319,E2 -13758.319} C_VEL
LIN {X 0,Y 346.519,Z 618.992,A -85,B 0,C 180,E1 -13760.663,E2 -13760.663} C_VEL
LIN {X 0,Y 346.227,Z 623.166,A -85,B 0,C 180,E1 -13763.005,E2 -13763.005} C_VEL
LIN {X 0,Y 346.124,Z 626.093,A -85,B 0,C 180,E1 -13765.341,E2 -13765.341} C_VEL
LIN {X 0,Y 346.075,Z 627.839,A -85,B 0,C 180,E1 -13767.672,E2 -13767.672} C_VEL
LIN {X 0,Y 346.162,Z 628.439,A -85,B 0,C 180,E1 -13770,E2 -13770} C_VEL
LIN {X 0,Y 346.075,Z 627.831,A -85,B 0,C 180,E1 -13772.328,E2 -13772.328} C_VEL
LIN {X 0,Y 346.117,Z 626.076,A -85,B 0,C 180,E1 -13774.659,E2 -13774.659} C_VEL
LIN {X 0,Y 346.224,Z 623.144,A -85,B 0,C 180,E1 -13776.995,E2 -13776.995} C_VEL
LIN {X 0,Y 346.514,Z 618.969,A -85,B 0,C 180,E1 -13779.338,E2 -13779.338} C_VEL
LIN {X 0,Y 347.107,Z 613.442,A -85,B 0,C 180,E1 -13781.681,E2 -13781.681} C_VEL
LIN {X 0,Y 347.897,Z 606.411,A -85,B 0,C 180,E1 -13784.029,E2 -13784.029} C_VEL
LIN {X 0,Y 349.11,Z 598.899,A -85,B 0,C 180,E1 -13786.069,E2 -13786.069} C_VEL
LIN {X 0,Y 350.562,Z 589.845,A -85,B 0,C 180,E1 -13788.103,E2 -13788.103} C_VEL
LIN {X 0,Y 352.481,Z 579.021,A -85,B 0,C 180,E1 -13790.108,E2 -13790.108} C_VEL
LIN {X 0,Y 354.407,Z 566.747,A -85,B 0,C 180,E1 -13791.98,E2 -13791.98} C_VEL
LIN {X 0,Y 356.498,Z 554.291,A -85,B 0,C 180,E1 -13793.528,E2 -13793.528} C_VEL
LIN {X 0,Y 358.374,Z 542.039,A -85,B 0,C 180,E1 -13794.782,E2 -13794.782} C_VEL
LIN {X 0,Y 360.243,Z 528.137,A -85,B 0,C 180,E1 -13795.939,E2 -13795.939} C_VEL
LIN {X 0,Y 361.788,Z 514.329,A -85,B 0,C 180,E1 -13796.849,E2 -13796.849} C_VEL
LIN {X 0,Y 363.178,Z 499.345,A -85,B 0,C 180,E1 -13797.594,E2 -13797.594} C_VEL
LIN {X 0,Y 364.239,Z 483.743,A -85,B 0,C 180,E1 -13798.132,E2 -13798.132} C_VEL
LIN {X 0,Y 365.407,Z 448.493,A -85,B 0,C 180,E1 -13798.854,E2 -13798.854} C_VEL
LIN {X 0,Y 367.643,Z 361.113,A -85,B 0,C 180,E1 -13800.584,E2 -13800.584} C_VEL
LIN {X 0,Y 363.278,Z 337.439,A -85,B 0,C 180,E1 -13801.523,E2 -13801.523} C_VEL
LIN {X 0,Y 354.884,Z 318.981,A -85,B 0,C 180,E1 -13802.783,E2 -13802.783} C_VEL
LIN {X 0,Y 353.373,Z 315.535,A -85,B 0,C 180,E1 -13803.038,E2 -13803.038} C_VEL
LIN {X 0,Y 350.125,Z 303.012,A -85,B 0,C 180,E1 -13806.177,E2 -13806.177} C_VEL
LIN {X 0,Y 347.717,Z 294.798,A -85,B 0,C 180,E1 -13808.397,E2 -13808.397} C_VEL
LIN {X 0,Y 347.738,Z 294.796,A -85,B 0,C 180,E1 -13811.831,E2 -13811.831} C_VEL
LIN {X 0,Y 347.697,Z 294.799,A -85,B 0,C 180,E1 -13815.027,E2 -13815.027} C_VEL
LIN {X 0,Y 347.734,Z 294.796,A -85,B 0,C 180,E1 -13818.398,E2 -13818.398} C_VEL
LIN {X 0,Y 347.746,Z 294.792,A -85,B 0,C 180,E1 -13822.677,E2 -13822.677} C_VEL
LIN {X 0,Y 347.74,Z 294.794,A -85,B 0,C 180,E1 -13825.956,E2 -13825.956} C_VEL
LIN {X 0,Y 347.73,Z 294.792,A -85,B 0,C 180,E1 -13829.65,E2 -13829.65} C_VEL
LIN {X 0,Y 347.733,Z 294.792,A -85,B 0,C 180,E1 -13833.6,E2 -13833.6} C_VEL
LIN {X 0,Y 347.742,Z 294.79,A -85,B 0,C 180,E1 -13836.159,E2 -13836.159} C_VEL
LIN {X 0,Y 347.788,Z 294.77,A -85,B 0,C 180,E1 -13839.908,E2 -13839.908} C_VEL
LIN {X 0,Y 347.821,Z 294.779,A -85,B 0,C 180,E1 -13843.568,E2 -13843.568} C_VEL
LIN {X 0,Y 347.875,Z 294.756,A -85,B 0,C 180,E1 -13847.16,E2 -13847.16} C_VEL
LIN {X 0,Y 347.922,Z 294.763,A -85,B 0,C 180,E1 -13850.7,E2 -13850.7} C_VEL
LIN {X 0,Y 348.035,Z 294.748,A -85,B 0,C 180,E1 -13854.205,E2 -13854.205} C_VEL
LIN {X 0,Y 348.178,Z 294.734,A -85,B 0,C 180,E1 -13857.686,E2 -13857.686} C_VEL
LIN {X 0,Y 348.105,Z 294.75,A -85,B 0,C 180,E1 -13861.157,E2 -13861.157} C_VEL
LIN {X 0,Y 348.182,Z 294.731,A -85,B 0,C 180,E1 -13862.314,E2 -13862.314} C_VEL
LIN {X 0,Y 348.062,Z 294.748,A -85,B 0,C 180,E1 -13866.959,E2 -13866.959} C_VEL
LIN {X 0,Y 347.885,Z 294.771,A -85,B 0,C 180,E1 -13870.476,E2 -13870.476} C_VEL
LIN {X 0,Y 347.89,Z 294.771,A -85,B 0,C 180,E1 -13874.15,E2 -13874.15} C_VEL
LIN {X 0,Y 347.82,Z 294.779,A -85,B 0,C 180,E1 -13878.259,E2 -13878.259} C_VEL
LIN {X 0,Y 347.759,Z 294.772,A -85,B 0,C 180,E1 -13881.627,E2 -13881.627} C_VEL
LIN {X 0,Y 347.791,Z 294.784,A -85,B 0,C 180,E1 -13885.11,E2 -13885.11} C_VEL
LIN {X 0,Y 347.791,Z 294.766,A -85,B 0,C 180,E1 -13887.696,E2 -13887.696} C_VEL
LIN {X 0,Y 347.742,Z 294.793,A -85,B 0,C 180,E1 -13890.349,E2 -13890.349} C_VEL
LIN {X 0,Y 347.741,Z 294.792,A -85,B 0,C 180,E1 -13894.044,E2 -13894.044} C_VEL
LIN {X 0,Y 347.754,Z 294.788,A -85,B 0,C 180,E1 -13897.322,E2 -13897.322} C_VEL
LIN {X 0,Y 347.726,Z 294.791,A -85,B 0,C 180,E1 -13900.298,E2 -13900.298} C_VEL
LIN {X 0,Y 347.718,Z 294.797,A -85,B 0,C 180,E1 -13903.409,E2 -13903.409} C_VEL
LIN {X 0,Y 347.721,Z 294.796,A -85,B 0,C 180,E1 -13906.687,E2 -13906.687} C_VEL
LIN {X 0,Y 347.744,Z 294.792,A -85,B 0,C 180,E1 -13910.174,E2 -13910.174} C_VEL
LIN {X 0,Y 347.759,Z 294.794,A -85,B 0,C 180,E1 -13912.68,E2 -13912.68} C_VEL
LIN {X 0,Y 347.801,Z 294.919,A -85,B 0,C 180,E1 -13915.324,E2 -13915.324} C_VEL
LIN {X 0,Y 349.058,Z 299.528,A -85,B 0,C 180,E1 -13916.581,E2 -13916.581} C_VEL
LIN {X 0,Y 358.713,Z 318.423,A -85,B 0,C 180,E1 -13918.041,E2 -13918.041} C_VEL
LIN {X 0,Y 366.779,Z 335.922,A -85,B 0,C 180,E1 -13919.223,E2 -13919.223} C_VEL
LIN {X 0,Y 368.085,Z 339.19,A -85,B 0,C 180,E1 -13919.417,E2 -13919.417} C_VEL
LIN {X 0,Y 365.875,Z 425.493,A -85,B 0,C 180,E1 -13921.128,E2 -13921.128} C_VEL
LIN {X 0,Y 364.622,Z 465.188,A -85,B 0,C 180,E1 -13921.939,E2 -13921.939} C_VEL
LIN {X 0,Y 363.773,Z 480.335,A -85,B 0,C 180,E1 -13922.47,E2 -13922.47} C_VEL
LIN {X 0,Y 362.568,Z 495.246,A -85,B 0,C 180,E1 -13923.217,E2 -13923.217} C_VEL
LIN {X 0,Y 361.061,Z 509.736,A -85,B 0,C 180,E1 -13924.182,E2 -13924.182} C_VEL
LIN {X 0,Y 359.304,Z 522.982,A -85,B 0,C 180,E1 -13925.286,E2 -13925.286} C_VEL
LIN {X 0,Y 357.427,Z 536.437,A -85,B 0,C 180,E1 -13926.69,E2 -13926.69} C_VEL
LIN {X 0,Y 355.534,Z 547.958,A -85,B 0,C 180,E1 -13928.144,E2 -13928.144} C_VEL
LIN {X 0,Y 353.898,Z 557.994,A -85,B 0,C 180,E1 -13929.664,E2 -13929.664} C_VEL
LIN {X 0,Y 352.162,Z 567.632,A -85,B 0,C 180,E1 -13931.38,E2 -13931.38} C_VEL
LIN {X 0,Y 350.506,Z 577.075,A -85,B 0,C 180,E1 -13933.398,E2 -13933.398} C_VEL
LIN {X 0,Y 349.098,Z 585.067,A -85,B 0,C 180,E1 -13935.465,E2 -13935.465} C_VEL
LIN {X 0,Y 348.329,Z 590.593,A -85,B 0,C 180,E1 -13937.177,E2 -13937.177} C_VEL
LIN {X 0,Y 347.367,Z 596.761,A -85,B 0,C 180,E1 -13939.509,E2 -13939.509} C_VEL
LIN {X 0,Y 346.79,Z 601.52,A -85,B 0,C 180,E1 -13941.845,E2 -13941.845} C_VEL
LIN {X 0,Y 346.438,Z 605.005,A -85,B 0,C 180,E1 -13944.179,E2 -13944.179} C_VEL
LIN {X 0,Y 346.221,Z 607.31,A -85,B 0,C 180,E1 -13946.509,E2 -13946.509} C_VEL
LIN {X 0,Y 346.153,Z 608.486,A -85,B 0,C 180,E1 -13948.837,E2 -13948.837} C_VEL
LIN {X 0,Y 346.153,Z 608.501,A -85,B 0,C 180,E1 -13951.163,E2 -13951.163} C_VEL
LIN {X 0,Y 346.216,Z 607.384,A -85,B 0,C 180,E1 -13953.491,E2 -13953.491} C_VEL
LIN {X 0,Y 346.415,Z 605.138,A -85,B 0,C 180,E1 -13955.822,E2 -13955.822} C_VEL
LIN {X 0,Y 346.756,Z 601.706,A -85,B 0,C 180,E1 -13958.156,E2 -13958.156} C_VEL
LIN {X 0,Y 347.328,Z 597.006,A -85,B 0,C 180,E1 -13960.492,E2 -13960.492} C_VEL
LIN {X 0,Y 348.299,Z 590.911,A -85,B 0,C 180,E1 -13962.824,E2 -13962.824} C_VEL
LIN {X 0,Y 349.454,Z 583.238,A -85,B 0,C 180,E1 -13965.156,E2 -13965.156} C_VEL
LIN {X 0,Y 350.885,Z 575.051,A -85,B 0,C 180,E1 -13967.183,E2 -13967.183} C_VEL
LIN {X 0,Y 352.616,Z 565.185,A -85,B 0,C 180,E1 -13969.199,E2 -13969.199} C_VEL
LIN {X 0,Y 354.39,Z 555.065,A -85,B 0,C 180,E1 -13970.913,E2 -13970.913} C_VEL
LIN {X 0,Y 356.336,Z 543.014,A -85,B 0,C 180,E1 -13972.618,E2 -13972.618} C_VEL
LIN {X 0,Y 358.041,Z 532.426,A -85,B 0,C 180,E1 -13973.855,E2 -13973.855} C_VEL
LIN {X 0,Y 358.099,Z 527.648,A -85,B 0,C 180,E1 -13974.409,E2 -13974.409} C_VEL
LIN {X 0,Y 356.626,Z 519.804,A -85,B 0,C 180,E1 -13975.358,E2 -13975.358} C_VEL
LIN {X 0,Y 355.131,Z 511.695,A -85,B 0,C 180,E1 -13976.238,E2 -13976.238} C_VEL
LIN {X 0,Y 355.132,Z 506.463,A -85,B 0,C 180,E1 -13976.676,E2 -13976.676} C_VEL
LIN {X 0,Y 356.568,Z 492.324,A -85,B 0,C 180,E1 -13977.578,E2 -13977.578} C_VEL
LIN {X 0,Y 357.74,Z 477.368,A -85,B 0,C 180,E1 -13978.29,E2 -13978.29} C_VEL
LIN {X 0,Y 358.652,Z 462.348,A -85,B 0,C 180,E1 -13978.771,E2 -13978.771} C_VEL
LIN {X 0,Y 362.084,Z 342.386,A -85,B 0,C 180,E1 -13981.187,E2 -13981.187} C_VEL
LIN {X 0,Y 361.753,Z 340.561,A -85,B 0,C 180,E1 -13981.26,E2 -13981.26} C_VEL
LIN {X 0,Y 353.003,Z 321.185,A -85,B 0,C 180,E1 -13982.591,E2 -13982.591} C_VEL
LIN {X 0,Y 343.518,Z 302.919,A -85,B 0,C 180,E1 -13984.066,E2 -13984.066} C_VEL
LIN {X 0,Y 341.763,Z 299.477,A -85,B 0,C 180,E1 -13984.367,E2 -13984.367} C_VEL
LIN {X 0,Y 340.726,Z 295.675,A -85,B 0,C 180,E1 -13985.549,E2 -13985.549} C_VEL
LIN {X 0,Y 340.707,Z 295.676,A -85,B 0,C 180,E1 -13988.385,E2 -13988.385} C_VEL
LIN {X 0,Y 340.695,Z 295.674,A -85,B 0,C 180,E1 -13992.044,E2 -13992.044} C_VEL
LIN {X 0,Y 340.647,Z 295.677,A -85,B 0,C 180,E1 -13996.226,E2 -13996.226} C_VEL
LIN {X 0,Y 340.682,Z 295.67,A -85,B 0,C 180,E1 -13999.752,E2 -13999.752} C_VEL
LIN {X 0,Y 340.696,Z 295.652,A -85,B 0,C 180,E1 -14003.257,E2 -14003.257} C_VEL
LIN {X 0,Y 340.685,Z 295.672,A -85,B 0,C 180,E1 -14006.152,E2 -14006.152} C_VEL
LIN {X 0,Y 340.722,Z 295.65,A -85,B 0,C 180,E1 -14010.327,E2 -14010.327} C_VEL
LIN {X 0,Y 340.771,Z 295.663,A -85,B 0,C 180,E1 -14013.017,E2 -14013.017} C_VEL
LIN {X 0,Y 340.744,Z 295.665,A -85,B 0,C 180,E1 -14015.637,E2 -14015.637} C_VEL
LIN {X 0,Y 340.724,Z 295.668,A -85,B 0,C 180,E1 -14019.473,E2 -14019.473} C_VEL
LIN {X 0,Y 340.784,Z 295.653,A -85,B 0,C 180,E1 -14021.98,E2 -14021.98} C_VEL
LIN {X 0,Y 340.844,Z 295.648,A -85,B 0,C 180,E1 -14025.716,E2 -14025.716} C_VEL
LIN {X 0,Y 340.837,Z 295.652,A -85,B 0,C 180,E1 -14029.305,E2 -14029.305} C_VEL
LIN {X 0,Y 341.031,Z 295.632,A -85,B 0,C 180,E1 -14032.897,E2 -14032.897} C_VEL
LIN {X 0,Y 341.146,Z 295.614,A -85,B 0,C 180,E1 -14037.638,E2 -14037.638} C_VEL
LIN {X 0,Y 341.224,Z 295.597,A -85,B 0,C 180,E1 -14040,E2 -14040} C_VEL
LIN {X 0,Y 341.116,Z 295.62,A -85,B 0,C 180,E1 -14042.361,E2 -14042.361} C_VEL
LIN {X 0,Y 341.009,Z 295.632,A -85,B 0,C 180,E1 -14047.103,E2 -14047.103} C_VEL
LIN {X 0,Y 340.835,Z 295.655,A -85,B 0,C 180,E1 -14050.695,E2 -14050.695} C_VEL
LIN {X 0,Y 340.854,Z 295.647,A -85,B 0,C 180,E1 -14054.325,E2 -14054.325} C_VEL
LIN {X 0,Y 340.776,Z 295.658,A -85,B 0,C 180,E1 -14058.44,E2 -14058.44} C_VEL
LIN {X 0,Y 340.71,Z 295.665,A -85,B 0,C 180,E1 -14061.842,E2 -14061.842} C_VEL
LIN {X 0,Y 340.667,Z 295.67,A -85,B 0,C 180,E1 -14065.673,E2 -14065.673} C_VEL
LIN {X 0,Y 340.674,Z 295.676,A -85,B 0,C 180,E1 -14068.326,E2 -14068.326} C_VEL
LIN {X 0,Y 340.685,Z 295.672,A -85,B 0,C 180,E1 -14071.046,E2 -14071.046} C_VEL
LIN {X 0,Y 340.707,Z 295.669,A -85,B 0,C 180,E1 -14075.28,E2 -14075.28} C_VEL
LIN {X 0,Y 340.685,Z 295.671,A -85,B 0,C 180,E1 -14078.383,E2 -14078.383} C_VEL
LIN {X 0,Y 340.687,Z 295.662,A -85,B 0,C 180,E1 -14082.045,E2 -14082.045} C_VEL
LIN {X 0,Y 340.644,Z 295.676,A -85,B 0,C 180,E1 -14086.228,E2 -14086.228} C_VEL
LIN {X 0,Y 340.662,Z 295.673,A -85,B 0,C 180,E1 -14088.688,E2 -14088.688} C_VEL
LIN {X 0,Y 340.695,Z 295.85,A -85,B 0,C 180,E1 -14090.978,E2 -14090.978} C_VEL
LIN {X 0,Y 343.869,Z 306.779,A -85,B 0,C 180,E1 -14093.96,E2 -14093.96} C_VEL
LIN {X 0,Y 346.163,Z 315.487,A -85,B 0,C 180,E1 -14096.181,E2 -14096.181} C_VEL
LIN {X 0,Y 355.897,Z 336.596,A -85,B 0,C 180,E1 -14097.712,E2 -14097.712} C_VEL
LIN {X 0,Y 357.719,Z 340.951,A -85,B 0,C 180,E1 -14097.996,E2 -14097.996} C_VEL
LIN {X 0,Y 361.511,Z 362.02,A -85,B 0,C 180,E1 -14098.847,E2 -14098.847} C_VEL
LIN {X 0,Y 359.297,Z 445.687,A -85,B 0,C 180,E1 -14100.531,E2 -14100.531} C_VEL
LIN {X 0,Y 358.125,Z 482.888,A -85,B 0,C 180,E1 -14101.303,E2 -14101.303} C_VEL
LIN {X 0,Y 357.094,Z 497.926,A -85,B 0,C 180,E1 -14101.814,E2 -14101.814} C_VEL
LIN {X 0,Y 355.584,Z 513.225,A -85,B 0,C 180,E1 -14102.564,E2 -14102.564} C_VEL
LIN {X 0,Y 353.908,Z 527.599,A -85,B 0,C 180,E1 -14103.513,E2 -14103.513} C_VEL
LIN {X 0,Y 351.911,Z 541.985,A -85,B 0,C 180,E1 -14104.731,E2 -14104.731} C_VEL
LIN {X 0,Y 349.739,Z 555.421,A -85,B 0,C 180,E1 -14106.146,E2 -14106.146} C_VEL
LIN {X 0,Y 347.61,Z 567.662,A -85,B 0,C 180,E1 -14107.723,E2 -14107.723} C_VEL
LIN {X 0,Y 345.667,Z 579.306,A -85,B 0,C 180,E1 -14109.555,E2 -14109.555} C_VEL
LIN {X 0,Y 343.753,Z 589.704,A -85,B 0,C 180,E1 -14111.525,E2 -14111.525} C_VEL
LIN {X 0,Y 342.205,Z 598.752,A -85,B 0,C 180,E1 -14113.598,E2 -14113.598} C_VEL
LIN {X 0,Y 340.997,Z 606.261,A -85,B 0,C 180,E1 -14115.681,E2 -14115.681} C_VEL
LIN {X 0,Y 340.092,Z 613.273,A -85,B 0,C 180,E1 -14118.074,E2 -14118.074} C_VEL
LIN {X 0,Y 339.444,Z 618.788,A -85,B 0,C 180,E1 -14120.466,E2 -14120.466} C_VEL
LIN {X 0,Y 339.145,Z 622.962,A -85,B 0,C 180,E1 -14122.858,E2 -14122.858} C_VEL
LIN {X 0,Y 339.029,Z 625.89,A -85,B 0,C 180,E1 -14125.244,E2 -14125.244} C_VEL
LIN {X 0,Y 338.989,Z 627.636,A -85,B 0,C 180,E1 -14127.624,E2 -14127.624} C_VEL
LIN {X 0,Y 339.065,Z 628.236,A -85,B 0,C 180,E1 -14130,E2 -14130} C_VEL
LIN {X 0,Y 338.989,Z 627.628,A -85,B 0,C 180,E1 -14132.376,E2 -14132.376} C_VEL
LIN {X 0,Y 339.021,Z 625.872,A -85,B 0,C 180,E1 -14134.756,E2 -14134.756} C_VEL
LIN {X 0,Y 339.143,Z 622.94,A -85,B 0,C 180,E1 -14137.142,E2 -14137.142} C_VEL
LIN {X 0,Y 339.44,Z 618.763,A -85,B 0,C 180,E1 -14139.534,E2 -14139.534} C_VEL
LIN {X 0,Y 340.091,Z 613.236,A -85,B 0,C 180,E1 -14141.926,E2 -14141.926} C_VEL
LIN {X 0,Y 340.911,Z 606.204,A -85,B 0,C 180,E1 -14144.322,E2 -14144.322} C_VEL
LIN {X 0,Y 342.214,Z 598.692,A -85,B 0,C 180,E1 -14146.402,E2 -14146.402} C_VEL
LIN {X 0,Y 343.767,Z 589.638,A -85,B 0,C 180,E1 -14148.474,E2 -14148.474} C_VEL
LIN {X 0,Y 345.686,Z 579.152,A -85,B 0,C 180,E1 -14150.457,E2 -14150.457} C_VEL
LIN {X 0,Y 347.596,Z 567.566,A -85,B 0,C 180,E1 -14152.277,E2 -14152.277} C_VEL
LIN {X 0,Y 349.749,Z 555.308,A -85,B 0,C 180,E1 -14153.853,E2 -14153.853} C_VEL
LIN {X 0,Y 351.688,Z 543.262,A -85,B 0,C 180,E1 -14155.128,E2 -14155.128} C_VEL
LIN {X 0,Y 353.667,Z 529.39,A -85,B 0,C 180,E1 -14156.328,E2 -14156.328} C_VEL
LIN {X 0,Y 355.332,Z 515.249,A -85,B 0,C 180,E1 -14157.297,E2 -14157.297} C_VEL
LIN {X 0,Y 356.763,Z 500.66,A -85,B 0,C 180,E1 -14158.054,E2 -14158.054} C_VEL
LIN {X 0,Y 357.888,Z 485.813,A -85,B 0,C 180,E1 -14158.597,E2 -14158.597} C_VEL
LIN {X 0,Y 358.649,Z 466.059,A -85,B 0,C 180,E1 -14159.051,E2 -14159.051} C_VEL
LIN {X 0,Y 361.572,Z 362.829,A -85,B 0,C 180,E1 -14161.11,E2 -14161.11} C_VEL
LIN {X 0,Y 357.521,Z 340.296,A -85,B 0,C 180,E1 -14162.019,E2 -14162.019} C_VEL
LIN {X 0,Y 349.363,Z 322.33,A -85,B 0,C 180,E1 -14163.283,E2 -14163.283} C_VEL
LIN {X 0,Y 346.058,Z 315.205,A -85,B 0,C 180,E1 -14163.848,E2 -14163.848} C_VEL
LIN {X 0,Y 343.13,Z 304.028,A -85,B 0,C 180,E1 -14166.742,E2 -14166.742} C_VEL
LIN {X 0,Y 340.662,Z 295.679,A -85,B 0,C 180,E1 -14169.063,E2 -14169.063} C_VEL
LIN {X 0,Y 340.668,Z 295.676,A -85,B 0,C 180,E1 -14172.904,E2 -14172.904} C_VEL
LIN {X 0,Y 340.667,Z 295.674,A -85,B 0,C 180,E1 -14177.094,E2 -14177.094} C_VEL
LIN {X 0,Y 340.648,Z 295.678,A -85,B 0,C 180,E1 -14180.24,E2 -14180.24} C_VEL
LIN {X 0,Y 340.699,Z 295.672,A -85,B 0,C 180,E1 -14183.56,E2 -14183.56} C_VEL
LIN {X 0,Y 340.684,Z 295.671,A -85,B 0,C 180,E1 -14186.153,E2 -14186.153} C_VEL
LIN {X 0,Y 340.713,Z 295.665,A -85,B 0,C 180,E1 -14190.034,E2 -14190.034} C_VEL
LIN {X 0,Y 340.709,Z 295.664,A -85,B 0,C 180,E1 -14193.012,E2 -14193.012} C_VEL
LIN {X 0,Y 340.695,Z 295.668,A -85,B 0,C 180,E1 -14196.925,E2 -14196.925} C_VEL
LIN {X 0,Y 340.724,Z 295.643,A -85,B 0,C 180,E1 -14200.73,E2 -14200.73} C_VEL
LIN {X 0,Y 340.807,Z 295.656,A -85,B 0,C 180,E1 -14204.45,E2 -14204.45} C_VEL
LIN {X 0,Y 340.833,Z 295.622,A -85,B 0,C 180,E1 -14208.1,E2 -14208.1} C_VEL
LIN {X 0,Y 340.97,Z 295.638,A -85,B 0,C 180,E1 -14211.704,E2 -14211.704} C_VEL
LIN {X 0,Y 341.01,Z 295.623,A -85,B 0,C 180,E1 -14214.085,E2 -14214.085} C_VEL
LIN {X 0,Y 341.115,Z 295.614,A -85,B 0,C 180,E1 -14217.639,E2 -14217.639} C_VEL
LIN {X 0,Y 341.077,Z 295.625,A -85,B 0,C 180,E1 -14221.181,E2 -14221.181} C_VEL
LIN {X 0,Y 341.12,Z 295.611,A -85,B 0,C 180,E1 -14222.362,E2 -14222.362} C_VEL
LIN {X 0,Y 341.009,Z 295.626,A -85,B 0,C 180,E1 -14227.103,E2 -14227.103} C_VEL
LIN {X 0,Y 340.837,Z 295.648,A -85,B 0,C 180,E1 -14230.695,E2 -14230.695} C_VEL
LIN {X 0,Y 340.855,Z 295.647,A -85,B 0,C 180,E1 -14234.325,E2 -14234.325} C_VEL
LIN {X 0,Y 340.777,Z 295.656,A -85,B 0,C 180,E1 -14238.441,E2 -14238.441} C_VEL
LIN {X 0,Y 340.71,Z 295.652,A -85,B 0,C 180,E1 -14241.842,E2 -14241.842} C_VEL
LIN {X 0,Y 340.75,Z 295.656,A -85,B 0,C 180,E1 -14245.666,E2 -14245.666} C_VEL
LIN {X 0,Y 340.715,Z 295.651,A -85,B 0,C 180,E1 -14248.322,E2 -14248.322} C_VEL
LIN {X 0,Y 340.69,Z 295.672,A -85,B 0,C 180,E1 -14251.046,E2 -14251.046} C_VEL
LIN {X 0,Y 340.709,Z 295.667,A -85,B 0,C 180,E1 -14255.28,E2 -14255.28} C_VEL
LIN {X 0,Y 340.703,Z 295.667,A -85,B 0,C 180,E1 -14258.387,E2 -14258.387} C_VEL
LIN {X 0,Y 340.694,Z 295.67,A -85,B 0,C 180,E1 -14262.046,E2 -14262.046} C_VEL
LIN {X 0,Y 340.647,Z 295.678,A -85,B 0,C 180,E1 -14266.228,E2 -14266.228} C_VEL
LIN {X 0,Y 340.685,Z 295.674,A -85,B 0,C 180,E1 -14269.754,E2 -14269.754} C_VEL
LIN {X 0,Y 340.702,Z 295.669,A -85,B 0,C 180,E1 -14273.259,E2 -14273.259} C_VEL
LIN {X 0,Y 340.723,Z 295.676,A -85,B 0,C 180,E1 -14274.632,E2 -14274.632} C_VEL
LIN {X 0,Y 341.86,Z 299.667,A -85,B 0,C 180,E1 -14275.778,E2 -14275.778} C_VEL
LIN {X 0,Y 351.776,Z 318.795,A -85,B 0,C 180,E1 -14277.336,E2 -14277.336} C_VEL
LIN {X 0,Y 360.889,Z 338.485,A -85,B 0,C 180,E1 -14278.718,E2 -14278.718} C_VEL
LIN {X 0,Y 361.955,Z 341.091,A -85,B 0,C 180,E1 -14278.88,E2 -14278.88} C_VEL
LIN {X 0,Y 359.638,Z 427.522,A -85,B 0,C 180,E1 -14280.619,E2 -14280.619} C_VEL
LIN {X 0,Y 358.391,Z 465.406,A -85,B 0,C 180,E1 -14281.407,E2 -14281.407} C_VEL
LIN {X 0,Y 357.494,Z 480.637,A -85,B 0,C 180,E1 -14281.948,E2 -14281.948} C_VEL
LIN {X 0,Y 356.275,Z 494.839,A -85,B 0,C 180,E1 -14282.662,E2 -14282.662} C_VEL
LIN {X 0,Y 354.939,Z 508.065,A -85,B 0,C 180,E1 -14283.545,E2 -14283.545} C_VEL
LIN {X 0,Y 353.076,Z 521.635,A -85,B 0,C 180,E1 -14284.663,E2 -14284.663} C_VEL
LIN {X 0,Y 351.09,Z 535.396,A -85,B 0,C 180,E1 -14286.087,E2 -14286.087} C_VEL
LIN {X 0,Y 349.184,Z 546.748,A -85,B 0,C 180,E1 -14287.518,E2 -14287.518} C_VEL
LIN {X 0,Y 347.247,Z 558.2,A -85,B 0,C 180,E1 -14289.257,E2 -14289.257} C_VEL
LIN {X 0,Y 345.421,Z 567.839,A -85,B 0,C 180,E1 -14291.002,E2 -14291.002} C_VEL
LIN {X 0,Y 343.661,Z 577.282,A -85,B 0,C 180,E1 -14293.058,E2 -14293.058} C_VEL
LIN {X 0,Y 342.075,Z 585.933,A -85,B 0,C 180,E1 -14295.361,E2 -14295.361} C_VEL
LIN {X 0,Y 341.038,Z 592.47,A -85,B 0,C 180,E1 -14297.504,E2 -14297.504} C_VEL
LIN {X 0,Y 340.166,Z 598.285,A -85,B 0,C 180,E1 -14299.886,E2 -14299.886} C_VEL
LIN {X 0,Y 339.753,Z 601.724,A -85,B 0,C 180,E1 -14301.675,E2 -14301.675} C_VEL
LIN {X 0,Y 339.365,Z 605.209,A -85,B 0,C 180,E1 -14304.057,E2 -14304.057} C_VEL
LIN {X 0,Y 339.148,Z 607.513,A -85,B 0,C 180,E1 -14306.436,E2 -14306.436} C_VEL
LIN {X 0,Y 339.055,Z 608.689,A -85,B 0,C 180,E1 -14308.812,E2 -14308.812} C_VEL
LIN {X 0,Y 339.055,Z 608.704,A -85,B 0,C 180,E1 -14311.188,E2 -14311.188} C_VEL
LIN {X 0,Y 339.143,Z 607.587,A -85,B 0,C 180,E1 -14313.564,E2 -14313.564} C_VEL
LIN {X 0,Y 339.346,Z 605.34,A -85,B 0,C 180,E1 -14315.944,E2 -14315.944} C_VEL
LIN {X 0,Y 339.723,Z 601.908,A -85,B 0,C 180,E1 -14318.326,E2 -14318.326} C_VEL
LIN {X 0,Y 340.32,Z 597.209,A -85,B 0,C 180,E1 -14320.711,E2 -14320.711} C_VEL
LIN {X 0,Y 341.357,Z 591.113,A -85,B 0,C 180,E1 -14323.089,E2 -14323.089} C_VEL
LIN {X 0,Y 342.562,Z 583.441,A -85,B 0,C 180,E1 -14325.468,E2 -14325.468} C_VEL
LIN {X 0,Y 344.087,Z 575.252,A -85,B 0,C 180,E1 -14327.533,E2 -14327.533} C_VEL
LIN {X 0,Y 345.886,Z 565.386,A -85,B 0,C 180,E1 -14329.588,E2 -14329.588} C_VEL
LIN {X 0,Y 347.909,Z 554.084,A -85,B 0,C 180,E1 -14331.523,E2 -14331.523} C_VEL
LIN {X 0,Y 349.96,Z 542.108,A -85,B 0,C 180,E1 -14333.21,E2 -14333.21} C_VEL
LIN {X 0,Y 351.978,Z 529.828,A -85,B 0,C 180,E1 -14334.633,E2 -14334.633} C_VEL
LIN {X 0,Y 353.909,Z 516.4,A -85,B 0,C 180,E1 -14335.904,E2 -14335.904} C_VEL
LIN {X 0,Y 355.132,Z 506.463,A -85,B 0,C 180,E1 -14336.676,E2 -14336.676} C_VEL
LIN {X 0,Y 354.939,Z 502.926,A -85,B 0,C 180,E1 -14336.978,E2 -14336.978} C_VEL
LIN {X 0,Y 350.896,Z 492.012,A -85,B 0,C 180,E1 -14338.095,E2 -14338.095} C_VEL
LIN {X 0,Y 350.643,Z 488.357,A -85,B 0,C 180,E1 -14338.345,E2 -14338.345} C_VEL
LIN {X 0,Y 351.832,Z 472.99,A -85,B 0,C 180,E1 -14339.013,E2 -14339.013} C_VEL
LIN {X 0,Y 352.658,Z 458.021,A -85,B 0,C 180,E1 -14339.429,E2 -14339.429} C_VEL
LIN {X 0,Y 355.97,Z 343.344,A -85,B 0,C 180,E1 -14341.766,E2 -14341.766} C_VEL
LIN {X 0,Y 348.636,Z 326.986,A -85,B 0,C 180,E1 -14342.914,E2 -14342.914} C_VEL
LIN {X 0,Y 340.324,Z 310.546,A -85,B 0,C 180,E1 -14344.242,E2 -14344.242} C_VEL
LIN {X 0,Y 334.5,Z 299.607,A -85,B 0,C 180,E1 -14345.251,E2 -14345.251} C_VEL
LIN {X 0,Y 333.675,Z 296.551,A -85,B 0,C 180,E1 -14346.224,E2 -14346.224} C_VEL
LIN {X 0,Y 333.643,Z 296.551,A -85,B 0,C 180,E1 -14349.191,E2 -14349.191} C_VEL
LIN {X 0,Y 333.629,Z 296.554,A -85,B 0,C 180,E1 -14352.499,E2 -14352.499} C_VEL
LIN {X 0,Y 333.592,Z 296.557,A -85,B 0,C 180,E1 -14355.954,E2 -14355.954} C_VEL
LIN {X 0,Y 333.642,Z 296.539,A -85,B 0,C 180,E1 -14359.315,E2 -14359.315} C_VEL
LIN {X 0,Y 333.657,Z 296.528,A -85,B 0,C 180,E1 -14363.168,E2 -14363.168} C_VEL
LIN {X 0,Y 333.63,Z 296.552,A -85,B 0,C 180,E1 -14366.791,E2 -14366.791} C_VEL
LIN {X 0,Y 333.671,Z 296.534,A -85,B 0,C 180,E1 -14371.024,E2 -14371.024} C_VEL
LIN {X 0,Y 333.692,Z 296.539,A -85,B 0,C 180,E1 -14373.75,E2 -14373.75} C_VEL
LIN {X 0,Y 333.657,Z 296.548,A -85,B 0,C 180,E1 -14376.409,E2 -14376.409} C_VEL
LIN {X 0,Y 333.679,Z 296.545,A -85,B 0,C 180,E1 -14380.306,E2 -14380.306} C_VEL
LIN {X 0,Y 333.748,Z 296.535,A -85,B 0,C 180,E1 -14384.112,E2 -14384.112} C_VEL
LIN {X 0,Y 333.783,Z 296.525,A -85,B 0,C 180,E1 -14386.608,E2 -14386.608} C_VEL
LIN {X 0,Y 333.811,Z 296.524,A -85,B 0,C 180,E1 -14390.303,E2 -14390.303} C_VEL
LIN {X 0,Y 333.992,Z 296.505,A -85,B 0,C 180,E1 -14393.96,E2 -14393.96} C_VEL
LIN {X 0,Y 334.082,Z 296.494,A -85,B 0,C 180,E1 -14397.589,E2 -14397.589} C_VEL
LIN {X 0,Y 334.177,Z 296.474,A -85,B 0,C 180,E1 -14400,E2 -14400} C_VEL
LIN {X 0,Y 334.057,Z 296.5,A -85,B 0,C 180,E1 -14402.411,E2 -14402.411} C_VEL
LIN {X 0,Y 333.988,Z 296.504,A -85,B 0,C 180,E1 -14406.039,E2 -14406.039} C_VEL
LIN {X 0,Y 333.809,Z 296.522,A -85,B 0,C 180,E1 -14409.697,E2 -14409.697} C_VEL
LIN {X 0,Y 333.783,Z 296.524,A -85,B 0,C 180,E1 -14413.392,E2 -14413.392} C_VEL
LIN {X 0,Y 333.709,Z 296.537,A -85,B 0,C 180,E1 -14417.148,E2 -14417.148} C_VEL
LIN {X 0,Y 333.661,Z 296.549,A -85,B 0,C 180,E1 -14419.695,E2 -14419.695} C_VEL
LIN {X 0,Y 333.633,Z 296.552,A -85,B 0,C 180,E1 -14423.593,E2 -14423.593} C_VEL
LIN {X 0,Y 333.659,Z 296.548,A -85,B 0,C 180,E1 -14427.606,E2 -14427.606} C_VEL
LIN {X 0,Y 333.649,Z 296.55,A -85,B 0,C 180,E1 -14430.367,E2 -14430.367} C_VEL
LIN {X 0,Y 333.629,Z 296.543,A -85,B 0,C 180,E1 -14433.209,E2 -14433.209} C_VEL
LIN {X 0,Y 333.665,Z 296.542,A -85,B 0,C 180,E1 -14436.14,E2 -14436.14} C_VEL
LIN {X 0,Y 333.594,Z 296.545,A -85,B 0,C 180,E1 -14439.2,E2 -14439.2} C_VEL
LIN {X 0,Y 333.622,Z 296.549,A -85,B 0,C 180,E1 -14442.5,E2 -14442.5} C_VEL
LIN {X 0,Y 333.588,Z 296.555,A -85,B 0,C 180,E1 -14445.955,E2 -14445.955} C_VEL
LIN {X 0,Y 333.596,Z 296.556,A -85,B 0,C 180,E1 -14449.325,E2 -14449.325} C_VEL
LIN {X 0,Y 333.626,Z 296.63,A -85,B 0,C 180,E1 -14450.242,E2 -14450.242} C_VEL
LIN {X 0,Y 336.929,Z 307.913,A -85,B 0,C 180,E1 -14453.423,E2 -14453.423} C_VEL
LIN {X 0,Y 338.844,Z 315.206,A -85,B 0,C 180,E1 -14455.347,E2 -14455.347} C_VEL
LIN {X 0,Y 348.466,Z 335.429,A -85,B 0,C 180,E1 -14456.914,E2 -14456.914} C_VEL
LIN {X 0,Y 351.922,Z 343.505,A -85,B 0,C 180,E1 -14457.469,E2 -14457.469} C_VEL
LIN {X 0,Y 355.422,Z 363.271,A -85,B 0,C 180,E1 -14458.285,E2 -14458.285} C_VEL
LIN {X 0,Y 353.031,Z 449.088,A -85,B 0,C 180,E1 -14460.038,E2 -14460.038} C_VEL
LIN {X 0,Y 351.92,Z 482.698,A -85,B 0,C 180,E1 -14460.749,E2 -14460.749} C_VEL
LIN {X 0,Y 350.855,Z 497.732,A -85,B 0,C 180,E1 -14461.267,E2 -14461.267} C_VEL
LIN {X 0,Y 349.291,Z 513.029,A -85,B 0,C 180,E1 -14462.027,E2 -14462.027} C_VEL
LIN {X 0,Y 347.663,Z 526.561,A -85,B 0,C 180,E1 -14462.927,E2 -14462.927} C_VEL
LIN {X 0,Y 345.696,Z 540.275,A -85,B 0,C 180,E1 -14464.082,E2 -14464.082} C_VEL
LIN {X 0,Y 343.676,Z 552.714,A -85,B 0,C 180,E1 -14465.377,E2 -14465.377} C_VEL
LIN {X 0,Y 341.55,Z 564.296,A -85,B 0,C 180,E1 -14466.826,E2 -14466.826} C_VEL
LIN {X 0,Y 339.453,Z 575.966,A -85,B 0,C 180,E1 -14468.596,E2 -14468.596} C_VEL
LIN {X 0,Y 337.545,Z 586.568,A -85,B 0,C 180,E1 -14470.541,E2 -14470.541} C_VEL
LIN {X 0,Y 335.764,Z 596.088,A -85,B 0,C 180,E1 -14472.647,E2 -14472.647} C_VEL
LIN {X 0,Y 334.387,Z 604.026,A -85,B 0,C 180,E1 -14474.769,E2 -14474.769} C_VEL
LIN {X 0,Y 333.303,Z 611.443,A -85,B 0,C 180,E1 -14477.209,E2 -14477.209} C_VEL
LIN {X 0,Y 332.505,Z 617.329,A -85,B 0,C 180,E1 -14479.65,E2 -14479.65} C_VEL
LIN {X 0,Y 332.229,Z 620.834,A -85,B 0,C 180,E1 -14481.485,E2 -14481.485} C_VEL
LIN {X 0,Y 332.01,Z 624.718,A -85,B 0,C 180,E1 -14484.208,E2 -14484.208} C_VEL
LIN {X 0,Y 331.946,Z 626.706,A -85,B 0,C 180,E1 -14486.358,E2 -14486.358} C_VEL
LIN {X 0,Y 331.92,Z 627.877,A -85,B 0,C 180,E1 -14488.787,E2 -14488.787} C_VEL
LIN {X 0,Y 331.92,Z 627.875,A -85,B 0,C 180,E1 -14491.213,E2 -14491.213} C_VEL
LIN {X 0,Y 331.944,Z 626.692,A -85,B 0,C 180,E1 -14493.642,E2 -14493.642} C_VEL
LIN {X 0,Y 331.993,Z 624.353,A -85,B 0,C 180,E1 -14496.076,E2 -14496.076} C_VEL
LIN {X 0,Y 332.222,Z 620.809,A -85,B 0,C 180,E1 -14498.516,E2 -14498.516} C_VEL
LIN {X 0,Y 332.64,Z 615.97,A -85,B 0,C 180,E1 -14500.961,E2 -14500.961} C_VEL
LIN {X 0,Y 333.501,Z 609.713,A -85,B 0,C 180,E1 -14503.403,E2 -14503.403} C_VEL
LIN {X 0,Y 334.561,Z 602.952,A -85,B 0,C 180,E1 -14505.535,E2 -14505.535} C_VEL
LIN {X 0,Y 335.97,Z 594.782,A -85,B 0,C 180,E1 -14507.656,E2 -14507.656} C_VEL
LIN {X 0,Y 337.868,Z 584.997,A -85,B 0,C 180,E1 -14509.755,E2 -14509.755} C_VEL
LIN {X 0,Y 339.736,Z 574.491,A -85,B 0,C 180,E1 -14511.63,E2 -14511.63} C_VEL
LIN {X 0,Y 341.591,Z 564.186,A -85,B 0,C 180,E1 -14513.171,E2 -14513.171} C_VEL
LIN {X 0,Y 343.861,Z 551.282,A -85,B 0,C 180,E1 -14514.77,E2 -14514.77} C_VEL
LIN {X 0,Y 345.921,Z 538.506,A -85,B 0,C 180,E1 -14516.062,E2 -14516.062} C_VEL
LIN {X 0,Y 347.782,Z 525.4,A -85,B 0,C 180,E1 -14517.138,E2 -14517.138} C_VEL
LIN {X 0,Y 349.446,Z 511.527,A -85,B 0,C 180,E1 -14518.041,E2 -14518.041} C_VEL
LIN {X 0,Y 350.828,Z 497.375,A -85,B 0,C 180,E1 -14518.736,E2 -14518.736} C_VEL
LIN {X 0,Y 351.876,Z 482.159,A -85,B 0,C 180,E1 -14519.255,E2 -14519.255} C_VEL
LIN {X 0,Y 354.722,Z 388.331,A -85,B 0,C 180,E1 -14521.182,E2 -14521.182} C_VEL
LIN {X 0,Y 355.363,Z 362.981,A -85,B 0,C 180,E1 -14521.707,E2 -14521.707} C_VEL
LIN {X 0,Y 351.549,Z 342.568,A -85,B 0,C 180,E1 -14522.571,E2 -14522.571} C_VEL
LIN {X 0,Y 344.016,Z 325.935,A -85,B 0,C 180,E1 -14523.776,E2 -14523.776} C_VEL
LIN {X 0,Y 338.821,Z 315.05,A -85,B 0,C 180,E1 -14524.65,E2 -14524.65} C_VEL
LIN {X 0,Y 335.725,Z 303.774,A -85,B 0,C 180,E1 -14527.691,E2 -14527.691} C_VEL
LIN {X 0,Y 333.619,Z 296.554,A -85,B 0,C 180,E1 -14529.778,E2 -14529.778} C_VEL
LIN {X 0,Y 333.623,Z 296.556,A -85,B 0,C 180,E1 -14532.498,E2 -14532.498} C_VEL
LIN {X 0,Y 333.589,Z 296.559,A -85,B 0,C 180,E1 -14535.954,E2 -14535.954} C_VEL
LIN {X 0,Y 333.596,Z 296.554,A -85,B 0,C 180,E1 -14539.324,E2 -14539.324} C_VEL
LIN {X 0,Y 333.653,Z 296.548,A -85,B 0,C 180,E1 -14543.168,E2 -14543.168} C_VEL
LIN {X 0,Y 333.665,Z 296.544,A -85,B 0,C 180,E1 -14545.34,E2 -14545.34} C_VEL
LIN {X 0,Y 333.621,Z 296.553,A -85,B 0,C 180,E1 -14548.221,E2 -14548.221} C_VEL
LIN {X 0,Y 333.644,Z 296.548,A -85,B 0,C 180,E1 -14551.022,E2 -14551.022} C_VEL
LIN {X 0,Y 333.655,Z 296.548,A -85,B 0,C 180,E1 -14555.085,E2 -14555.085} C_VEL
LIN {X 0,Y 333.654,Z 296.543,A -85,B 0,C 180,E1 -14559.018,E2 -14559.018} C_VEL
LIN {X 0,Y 333.731,Z 296.513,A -85,B 0,C 180,E1 -14561.586,E2 -14561.586} C_VEL
LIN {X 0,Y 333.799,Z 296.527,A -85,B 0,C 180,E1 -14565.577,E2 -14565.577} C_VEL
LIN {X 0,Y 333.801,Z 296.498,A -85,B 0,C 180,E1 -14569.077,E2 -14569.077} C_VEL
LIN {X 0,Y 333.952,Z 296.511,A -85,B 0,C 180,E1 -14572.746,E2 -14572.746} C_VEL
LIN {X 0,Y 333.772,Z 296.527,A -85,B 0,C 180,E1 -14575.169,E2 -14575.169} C_VEL
LIN {X 0,Y 334.056,Z 296.494,A -85,B 0,C 180,E1 -14577.589,E2 -14577.589} C_VEL
LIN {X 0,Y 334.048,Z 296.5,A -85,B 0,C 180,E1 -14581.206,E2 -14581.206} C_VEL
LIN {X 0,Y 334.06,Z 296.491,A -85,B 0,C 180,E1 -14582.412,E2 -14582.412} C_VEL
LIN {X 0,Y 333.958,Z 296.503,A -85,B 0,C 180,E1 -14586.587,E2 -14586.587} C_VEL
LIN {X 0,Y 333.81,Z 296.526,A -85,B 0,C 180,E1 -14589.697,E2 -14589.697} C_VEL
LIN {X 0,Y 333.783,Z 296.532,A -85,B 0,C 180,E1 -14593.392,E2 -14593.392} C_VEL
LIN {X 0,Y 333.71,Z 296.543,A -85,B 0,C 180,E1 -14597.148,E2 -14597.148} C_VEL
LIN {X 0,Y 333.662,Z 296.524,A -85,B 0,C 180,E1 -14599.695,E2 -14599.695} C_VEL
LIN {X 0,Y 333.662,Z 296.548,A -85,B 0,C 180,E1 -14603.591,E2 -14603.591} C_VEL
LIN {X 0,Y 333.692,Z 296.529,A -85,B 0,C 180,E1 -14606.25,E2 -14606.25} C_VEL
LIN {X 0,Y 333.68,Z 296.534,A -85,B 0,C 180,E1 -14608.975,E2 -14608.975} C_VEL
LIN {X 0,Y 333.636,Z 296.546,A -85,B 0,C 180,E1 -14612.588,E2 -14612.588} C_VEL
LIN {X 0,Y 333.668,Z 296.545,A -85,B 0,C 180,E1 -14616.14,E2 -14616.14} C_VEL
LIN {X 0,Y 333.641,Z 296.548,A -85,B 0,C 180,E1 -14619.193,E2 -14619.193} C_VEL
LIN {X 0,Y 333.627,Z 296.549,A -85,B 0,C 180,E1 -14622.501,E2 -14622.501} C_VEL
LIN {X 0,Y 333.592,Z 296.557,A -85,B 0,C 180,E1 -14625.956,E2 -14625.956} C_VEL
LIN {X 0,Y 333.644,Z 296.553,A -85,B 0,C 180,E1 -14629.316,E2 -14629.316} C_VEL
LIN {X 0,Y 333.662,Z 296.547,A -85,B 0,C 180,E1 -14633.169,E2 -14633.169} C_VEL
LIN {X 0,Y 333.706,Z 296.597,A -85,B 0,C 180,E1 -14633.957,E2 -14633.957} C_VEL
LIN {X 0,Y 334.667,Z 300.033,A -85,B 0,C 180,E1 -14634.939,E2 -14634.939} C_VEL
LIN {X 0,Y 344.55,Z 318.62,A -85,B 0,C 180,E1 -14636.551,E2 -14636.551} C_VEL
LIN {X 0,Y 354.252,Z 339.23,A -85,B 0,C 180,E1 -14638.075,E2 -14638.075} C_VEL
LIN {X 0,Y 355.915,Z 343.233,A -85,B 0,C 180,E1 -14638.336,E2 -14638.336} C_VEL
LIN {X 0,Y 353.031,Z 442.76,A -85,B 0,C 180,E1 -14640.359,E2 -14640.359} C_VEL
LIN {X 0,Y 352.122,Z 466.764,A -85,B 0,C 180,E1 -14640.89,E2 -14640.89} C_VEL
LIN {X 0,Y 351.129,Z 482.28,A -85,B 0,C 180,E1 -14641.47,E2 -14641.47} C_VEL
LIN {X 0,Y 349.86,Z 496.415,A -85,B 0,C 180,E1 -14642.216,E2 -14642.216} C_VEL
LIN {X 0,Y 348.355,Z 510.153,A -85,B 0,C 180,E1 -14643.167,E2 -14643.167} C_VEL
LIN {X 0,Y 346.447,Z 523.399,A -85,B 0,C 180,E1 -14644.304,E2 -14644.304} C_VEL
LIN {X 0,Y 344.395,Z 536.852,A -85,B 0,C 180,E1 -14645.753,E2 -14645.753} C_VEL
LIN {X 0,Y 342.32,Z 548.694,A -85,B 0,C 180,E1 -14647.303,E2 -14647.303} C_VEL
LIN {X 0,Y 340.237,Z 560.175,A -85,B 0,C 180,E1 -14649.126,E2 -14649.126} C_VEL
LIN {X 0,Y 338.12,Z 570.969,A -85,B 0,C 180,E1 -14651.206,E2 -14651.206} C_VEL
LIN {X 0,Y 336.378,Z 579.926,A -85,B 0,C 180,E1 -14653.305,E2 -14653.305} C_VEL
LIN {X 0,Y 335.006,Z 587.343,A -85,B 0,C 180,E1 -14655.42,E2 -14655.42} C_VEL
LIN {X 0,Y 334.087,Z 592.675,A -85,B 0,C 180,E1 -14657.24,E2 -14657.24} C_VEL
LIN {X 0,Y 333.148,Z 598.49,A -85,B 0,C 180,E1 -14659.671,E2 -14659.671} C_VEL
LIN {X 0,Y 332.709,Z 601.929,A -85,B 0,C 180,E1 -14661.497,E2 -14661.497} C_VEL
LIN {X 0,Y 332.308,Z 605.413,A -85,B 0,C 180,E1 -14663.93,E2 -14663.93} C_VEL
LIN {X 0,Y 332.077,Z 607.716,A -85,B 0,C 180,E1 -14666.36,E2 -14666.36} C_VEL
LIN {X 0,Y 331.96,Z 608.892,A -85,B 0,C 180,E1 -14668.787,E2 -14668.787} C_VEL
LIN {X 0,Y 331.96,Z 608.906,A -85,B 0,C 180,E1 -14671.213,E2 -14671.213} C_VEL
LIN {X 0,Y 332.072,Z 607.789,A -85,B 0,C 180,E1 -14673.64,E2 -14673.64} C_VEL
LIN {X 0,Y 332.312,Z 605.292,A -85,B 0,C 180,E1 -14676.282,E2 -14676.282} C_VEL
LIN {X 0,Y 332.808,Z 601.057,A -85,B 0,C 180,E1 -14679.113,E2 -14679.113} C_VEL
LIN {X 0,Y 333.511,Z 596.003,A -85,B 0,C 180,E1 -14681.548,E2 -14681.548} C_VEL
LIN {X 0,Y 334.692,Z 589.524,A -85,B 0,C 180,E1 -14683.974,E2 -14683.974} C_VEL
LIN {X 0,Y 335.901,Z 582.534,A -85,B 0,C 180,E1 -14686.094,E2 -14686.094} C_VEL
LIN {X 0,Y 337.522,Z 574.117,A -85,B 0,C 180,E1 -14688.199,E2 -14688.199} C_VEL
LIN {X 0,Y 339.463,Z 563.977,A -85,B 0,C 180,E1 -14690.29,E2 -14690.29} C_VEL
LIN {X 0,Y 341.449,Z 553.101,A -85,B 0,C 180,E1 -14692.145,E2 -14692.145} C_VEL
LIN {X 0,Y 343.65,Z 541.139,A -85,B 0,C 180,E1 -14693.822,E2 -14693.822} C_VEL
LIN {X 0,Y 345.695,Z 528.623,A -85,B 0,C 180,E1 -14695.272,E2 -14695.272} C_VEL
LIN {X 0,Y 347.757,Z 514.866,A -85,B 0,C 180,E1 -14696.559,E2 -14696.559} C_VEL
LIN {X 0,Y 349.536,Z 500.638,A -85,B 0,C 180,E1 -14697.616,E2 -14697.616} C_VEL
LIN {X 0,Y 350.643,Z 488.357,A -85,B 0,C 180,E1 -14698.345,E2 -14698.345} C_VEL
LIN {X 0,Y 350.598,Z 482.797,A -85,B 0,C 180,E1 -14698.67,E2 -14698.67} C_VEL
LIN {X 0,Y 348.799,Z 473.753,A -85,B 0,C 180,E1 -14699.264,E2 -14699.264} C_VEL
LIN {X 0,Y 346.861,Z 464.581,A -85,B 0,C 180,E1 -14699.791,E2 -14699.791} C_VEL
LIN {X 0,Y 346.478,Z 458.824,A -85,B 0,C 180,E1 -14699.99,E2 -14699.99} C_VEL
LIN {X 0,Y 349.927,Z 345.36,A -85,B 0,C 180,E1 -14702.337,E2 -14702.337} C_VEL
LIN {X 0,Y 341.632,Z 327.042,A -85,B 0,C 180,E1 -14703.681,E2 -14703.681} C_VEL
LIN {X 0,Y 331.601,Z 307.705,A -85,B 0,C 180,E1 -14705.355,E2 -14705.355} C_VEL
LIN {X 0,Y 327.375,Z 299.931,A -85,B 0,C 180,E1 -14706.115,E2 -14706.115} C_VEL
LIN {X 0,Y 326.613,Z 297.424,A -85,B 0,C 180,E1 -14706.926,E2 -14706.926} C_VEL
LIN {X 0,Y 326.588,Z 297.42,A -85,B 0,C 180,E1 -14710.208,E2 -14710.208} C_VEL
LIN {X 0,Y 326.558,Z 297.434,A -85,B 0,C 180,E1 -14713.525,E2 -14713.525} C_VEL
LIN {X 0,Y 326.571,Z 297.422,A -85,B 0,C 180,E1 -14717.027,E2 -14717.027} C_VEL
LIN {X 0,Y 326.605,Z 297.428,A -85,B 0,C 180,E1 -14720.772,E2 -14720.772} C_VEL
LIN {X 0,Y 326.604,Z 297.414,A -85,B 0,C 180,E1 -14724.479,E2 -14724.479} C_VEL
LIN {X 0,Y 326.601,Z 297.419,A -85,B 0,C 180,E1 -14727.455,E2 -14727.455} C_VEL
LIN {X 0,Y 326.62,Z 297.405,A -85,B 0,C 180,E1 -14730.337,E2 -14730.337} C_VEL
LIN {X 0,Y 326.65,Z 297.421,A -85,B 0,C 180,E1 -14733.139,E2 -14733.139} C_VEL
LIN {X 0,Y 326.636,Z 297.422,A -85,B 0,C 180,E1 -14735.87,E2 -14735.87} C_VEL
LIN {X 0,Y 326.622,Z 297.423,A -85,B 0,C 180,E1 -14739.862,E2 -14739.862} C_VEL
LIN {X 0,Y 326.655,Z 297.412,A -85,B 0,C 180,E1 -14742.47,E2 -14742.47} C_VEL
LIN {X 0,Y 326.747,Z 297.401,A -85,B 0,C 180,E1 -14746.314,E2 -14746.314} C_VEL
LIN {X 0,Y 326.773,Z 297.403,A -85,B 0,C 180,E1 -14750.092,E2 -14750.092} C_VEL
LIN {X 0,Y 326.948,Z 297.382,A -85,B 0,C 180,E1 -14753.83,E2 -14753.83} C_VEL
LIN {X 0,Y 327.023,Z 297.374,A -85,B 0,C 180,E1 -14757.536,E2 -14757.536} C_VEL
LIN {X 0,Y 327.13,Z 297.352,A -85,B 0,C 180,E1 -14760,E2 -14760} C_VEL
LIN {X 0,Y 327,Z 297.379,A -85,B 0,C 180,E1 -14762.463,E2 -14762.463} C_VEL
LIN {X 0,Y 326.942,Z 297.382,A -85,B 0,C 180,E1 -14766.17,E2 -14766.17} C_VEL
LIN {X 0,Y 326.772,Z 297.399,A -85,B 0,C 180,E1 -14769.907,E2 -14769.907} C_VEL
LIN {X 0,Y 326.747,Z 297.4,A -85,B 0,C 180,E1 -14773.686,E2 -14773.686} C_VEL
LIN {X 0,Y 326.654,Z 297.415,A -85,B 0,C 180,E1 -14777.53,E2 -14777.53} C_VEL
LIN {X 0,Y 326.605,Z 297.423,A -85,B 0,C 180,E1 -14781.457,E2 -14781.457} C_VEL
LIN {X 0,Y 326.594,Z 297.423,A -85,B 0,C 180,E1 -14785.492,E2 -14785.492} C_VEL
LIN {X 0,Y 326.608,Z 297.427,A -85,B 0,C 180,E1 -14789.664,E2 -14789.664} C_VEL
LIN {X 0,Y 326.609,Z 297.417,A -85,B 0,C 180,E1 -14792.946,E2 -14792.946} C_VEL
LIN {X 0,Y 326.602,Z 297.426,A -85,B 0,C 180,E1 -14795.521,E2 -14795.521} C_VEL
LIN {X 0,Y 326.566,Z 297.42,A -85,B 0,C 180,E1 -14799.219,E2 -14799.219} C_VEL
LIN {X 0,Y 326.567,Z 297.432,A -85,B 0,C 180,E1 -14802.972,E2 -14802.972} C_VEL
LIN {X 0,Y 326.566,Z 297.431,A -85,B 0,C 180,E1 -14807.03,E2 -14807.03} C_VEL
LIN {X 0,Y 326.581,Z 297.539,A -85,B 0,C 180,E1 -14809.505,E2 -14809.505} C_VEL
LIN {X 0,Y 329.763,Z 308.242,A -85,B 0,C 180,E1 -14812.635,E2 -14812.635} C_VEL
LIN {X 0,Y 331.694,Z 315.183,A -85,B 0,C 180,E1 -14814.494,E2 -14814.494} C_VEL
LIN {X 0,Y 341.235,Z 334.887,A -85,B 0,C 180,E1 -14816.111,E2 -14816.111} C_VEL
LIN {X 0,Y 346.259,Z 346.711,A -85,B 0,C 180,E1 -14816.951,E2 -14816.951} C_VEL
LIN {X 0,Y 349.38,Z 364.329,A -85,B 0,C 180,E1 -14817.701,E2 -14817.701} C_VEL
LIN {X 0,Y 346.649,Z 457.543,A -85,B 0,C 180,E1 -14819.631,E2 -14819.631} C_VEL
LIN {X 0,Y 345.685,Z 483.649,A -85,B 0,C 180,E1 -14820.21,E2 -14820.21} C_VEL
LIN {X 0,Y 344.571,Z 498.302,A -85,B 0,C 180,E1 -14820.734,E2 -14820.734} C_VEL
LIN {X 0,Y 343.015,Z 512.831,A -85,B 0,C 180,E1 -14821.469,E2 -14821.469} C_VEL
LIN {X 0,Y 341.18,Z 527.465,A -85,B 0,C 180,E1 -14822.468,E2 -14822.468} C_VEL
LIN {X 0,Y 339.055,Z 541.585,A -85,B 0,C 180,E1 -14823.701,E2 -14823.701} C_VEL
LIN {X 0,Y 336.739,Z 555.02,A -85,B 0,C 180,E1 -14825.165,E2 -14825.165} C_VEL
LIN {X 0,Y 334.427,Z 567.259,A -85,B 0,C 180,E1 -14826.795,E2 -14826.795} C_VEL
LIN {X 0,Y 332.134,Z 579.152,A -85,B 0,C 180,E1 -14828.733,E2 -14828.733} C_VEL
LIN {X 0,Y 330.192,Z 589.298,A -85,B 0,C 180,E1 -14830.737,E2 -14830.737} C_VEL
LIN {X 0,Y 328.453,Z 598.345,A -85,B 0,C 180,E1 -14832.89,E2 -14832.89} C_VEL
LIN {X 0,Y 327.041,Z 606.452,A -85,B 0,C 180,E1 -14835.247,E2 -14835.247} C_VEL
LIN {X 0,Y 326.09,Z 612.866,A -85,B 0,C 180,E1 -14837.554,E2 -14837.554} C_VEL
LIN {X 0,Y 325.345,Z 618.381,A -85,B 0,C 180,E1 -14840.049,E2 -14840.049} C_VEL
LIN {X 0,Y 324.976,Z 622.555,A -85,B 0,C 180,E1 -14842.545,E2 -14842.545} C_VEL
LIN {X 0,Y 324.854,Z 625.484,A -85,B 0,C 180,E1 -14845.036,E2 -14845.036} C_VEL
LIN {X 0,Y 324.825,Z 627.231,A -85,B 0,C 180,E1 -14847.52,E2 -14847.52} C_VEL
LIN {X 0,Y 324.872,Z 627.83,A -85,B 0,C 180,E1 -14850,E2 -14850} C_VEL
LIN {X 0,Y 324.825,Z 627.223,A -85,B 0,C 180,E1 -14852.48,E2 -14852.48} C_VEL
LIN {X 0,Y 324.846,Z 625.465,A -85,B 0,C 180,E1 -14854.964,E2 -14854.964} C_VEL
LIN {X 0,Y 324.973,Z 622.53,A -85,B 0,C 180,E1 -14857.455,E2 -14857.455} C_VEL
LIN {X 0,Y 325.343,Z 618.353,A -85,B 0,C 180,E1 -14859.951,E2 -14859.951} C_VEL
LIN {X 0,Y 326.089,Z 612.824,A -85,B 0,C 180,E1 -14862.446,E2 -14862.446} C_VEL
LIN {X 0,Y 327.073,Z 605.792,A -85,B 0,C 180,E1 -14864.942,E2 -14864.942} C_VEL
LIN {X 0,Y 328.711,Z 597.055,A -85,B 0,C 180,E1 -14867.417,E2 -14867.417} C_VEL
LIN {X 0,Y 330.206,Z 589.224,A -85,B 0,C 180,E1 -14869.262,E2 -14869.262} C_VEL
LIN {X 0,Y 332.214,Z 578.854,A -85,B 0,C 180,E1 -14871.302,E2 -14871.302} C_VEL
LIN {X 0,Y 334.413,Z 567.152,A -85,B 0,C 180,E1 -14873.206,E2 -14873.206} C_VEL
LIN {X 0,Y 336.716,Z 554.892,A -85,B 0,C 180,E1 -14874.837,E2 -14874.837} C_VEL
LIN {X 0,Y 339.054,Z 541.414,A -85,B 0,C 180,E1 -14876.299,E2 -14876.299} C_VEL
LIN {X 0,Y 341.19,Z 527.201,A -85,B 0,C 180,E1 -14877.535,E2 -14877.535} C_VEL
LIN {X 0,Y 343.041,Z 512.567,A -85,B 0,C 180,E1 -14878.529,E2 -14878.529} C_VEL
LIN {X 0,Y 344.536,Z 497.947,A -85,B 0,C 180,E1 -14879.269,E2 -14879.269} C_VEL
LIN {X 0,Y 345.713,Z 481.942,A -85,B 0,C 180,E1 -14879.829,E2 -14879.829} C_VEL
LIN {X 0,Y 348.792,Z 384.262,A -85,B 0,C 180,E1 -14881.865,E2 -14881.865} C_VEL
LIN {X 0,Y 349.313,Z 364.13,A -85,B 0,C 180,E1 -14882.289,E2 -14882.289} C_VEL
LIN {X 0,Y 345.989,Z 345.679,A -85,B 0,C 180,E1 -14883.081,E2 -14883.081} C_VEL
LIN {X 0,Y 337.551,Z 327.048,A -85,B 0,C 180,E1 -14884.479,E2 -14884.479} C_VEL
LIN {X 0,Y 331.512,Z 314.699,A -85,B 0,C 180,E1 -14885.553,E2 -14885.553} C_VEL
LIN {X 0,Y 328.353,Z 303.521,A -85,B 0,C 180,E1 -14888.692,E2 -14888.692} C_VEL
LIN {X 0,Y 326.572,Z 297.436,A -85,B 0,C 180,E1 -14890.521,E2 -14890.521} C_VEL
LIN {X 0,Y 326.555,Z 297.434,A -85,B 0,C 180,E1 -14893.525,E2 -14893.525} C_VEL
LIN {X 0,Y 326.567,Z 297.431,A -85,B 0,C 180,E1 -14897.028,E2 -14897.028} C_VEL
LIN {X 0,Y 326.574,Z 297.429,A -85,B 0,C 180,E1 -14901.385,E2 -14901.385} C_VEL
LIN {X 0,Y 326.61,Z 297.422,A -85,B 0,C 180,E1 -14904.851,E2 -14904.851} C_VEL
LIN {X 0,Y 326.6,Z 297.422,A -85,B 0,C 180,E1 -14907.455,E2 -14907.455} C_VEL
LIN {X 0,Y 326.607,Z 297.423,A -85,B 0,C 180,E1 -14910.336,E2 -14910.336} C_VEL
LIN {X 0,Y 326.593,Z 297.428,A -85,B 0,C 180,E1 -14914.508,E2 -14914.508} C_VEL
LIN {X 0,Y 326.605,Z 297.423,A -85,B 0,C 180,E1 -14918.543,E2 -14918.543} C_VEL
LIN {X 0,Y 326.654,Z 297.404,A -85,B 0,C 180,E1 -14922.47,E2 -14922.47} C_VEL
LIN {X 0,Y 326.746,Z 297.4,A -85,B 0,C 180,E1 -14926.314,E2 -14926.314} C_VEL
LIN {X 0,Y 326.77,Z 297.387,A -85,B 0,C 180,E1 -14930.093,E2 -14930.093} C_VEL
LIN {X 0,Y 326.937,Z 297.378,A -85,B 0,C 180,E1 -14933.83,E2 -14933.83} C_VEL
LIN {X 0,Y 326.999,Z 297.373,A -85,B 0,C 180,E1 -14937.537,E2 -14937.537} C_VEL
LIN {X 0,Y 327.018,Z 297.375,A -85,B 0,C 180,E1 -14941.232,E2 -14941.232} C_VEL
LIN {X 0,Y 326.754,Z 297.406,A -85,B 0,C 180,E1 -14943.7,E2 -14943.7} C_VEL
LIN {X 0,Y 326.917,Z 297.38,A -85,B 0,C 180,E1 -14946.578,E2 -14946.578} C_VEL
LIN {X 0,Y 326.773,Z 297.402,A -85,B 0,C 180,E1 -14949.908,E2 -14949.908} C_VEL
LIN {X 0,Y 326.747,Z 297.406,A -85,B 0,C 180,E1 -14953.686,E2 -14953.686} C_VEL
LIN {X 0,Y 326.655,Z 297.418,A -85,B 0,C 180,E1 -14957.53,E2 -14957.53} C_VEL
LIN {X 0,Y 326.609,Z 297.402,A -85,B 0,C 180,E1 -14961.457,E2 -14961.457} C_VEL
LIN {X 0,Y 326.642,Z 297.414,A -85,B 0,C 180,E1 -14965.488,E2 -14965.488} C_VEL
LIN {X 0,Y 326.638,Z 297.403,A -85,B 0,C 180,E1 -14968.252,E2 -14968.252} C_VEL
LIN {X 0,Y 326.583,Z 297.428,A -85,B 0,C 180,E1 -14971.096,E2 -14971.096} C_VEL
LIN {X 0,Y 326.6,Z 297.426,A -85,B 0,C 180,E1 -14974.02,E2 -14974.02} C_VEL
LIN {X 0,Y 326.62,Z 297.42,A -85,B 0,C 180,E1 -14977.239,E2 -14977.239} C_VEL
LIN {X 0,Y 326.573,Z 297.432,A -85,B 0,C 180,E1 -14981.132,E2 -14981.132} C_VEL
LIN {X 0,Y 326.523,Z 297.435,A -85,B 0,C 180,E1 -14984.744,E2 -14984.744} C_VEL
LIN {X 0,Y 326.572,Z 297.432,A -85,B 0,C 180,E1 -14988.155,E2 -14988.155} C_VEL
LIN {X 0,Y 326.595,Z 297.418,A -85,B 0,C 180,E1 -14991.389,E2 -14991.389} C_VEL
LIN {X 0,Y 326.657,Z 297.61,A -85,B 0,C 180,E1 -14993.265,E2 -14993.265} C_VEL
LIN {X 0,Y 327.392,Z 300.123,A -85,B 0,C 180,E1 -14994.035,E2 -14994.035} C_VEL
LIN {X 0,Y 338.043,Z 319.884,A -85,B 0,C 180,E1 -14995.845,E2 -14995.845} C_VEL
LIN {X 0,Y 347.065,Z 338.757,A -85,B 0,C 180,E1 -14997.314,E2 -14997.314} C_VEL
LIN {X 0,Y 349.811,Z 345.109,A -85,B 0,C 180,E1 -14997.757,E2 -14997.757} C_VEL
LIN {X 0,Y 347.126,Z 435.841,A -85,B 0,C 180,E1 -14999.635,E2 -14999.635} C_VEL
LIN {X 0,Y 346.012,Z 465.843,A -85,B 0,C 180,E1 -15000.283,E2 -15000.283} C_VEL
LIN {X 0,Y 345.016,Z 481.258,A -85,B 0,C 180,E1 -15000.849,E2 -15000.849} C_VEL
LIN {X 0,Y 343.723,Z 495.358,A -85,B 0,C 180,E1 -15001.582,E2 -15001.582} C_VEL
LIN {X 0,Y 342.283,Z 508.485,A -85,B 0,C 180,E1 -15002.486,E2 -15002.486} C_VEL
LIN {X 0,Y 340.29,Z 522.052,A -85,B 0,C 180,E1 -15003.639,E2 -15003.639} C_VEL
LIN {X 0,Y 338.13,Z 535.812,A -85,B 0,C 180,E1 -15005.11,E2 -15005.11} C_VEL
LIN {X 0,Y 336.038,Z 547.163,A -85,B 0,C 180,E1 -15006.587,E2 -15006.587} C_VEL
LIN {X 0,Y 334.326,Z 556.841,A -85,B 0,C 180,E1 -15008.092,E2 -15008.092} C_VEL
LIN {X 0,Y 332.263,Z 566.776,A -85,B 0,C 180,E1 -15009.897,E2 -15009.897} C_VEL
LIN {X 0,Y 330.317,Z 576.472,A -85,B 0,C 180,E1 -15012.031,E2 -15012.031} C_VEL
LIN {X 0,Y 328.569,Z 584.846,A -85,B 0,C 180,E1 -15014.268,E2 -15014.268} C_VEL
LIN {X 0,Y 327.484,Z 591.21,A -85,B 0,C 180,E1 -15016.346,E2 -15016.346} C_VEL
LIN {X 0,Y 326.361,Z 597.377,A -85,B 0,C 180,E1 -15018.825,E2 -15018.825} C_VEL
LIN {X 0,Y 325.664,Z 602.134,A -85,B 0,C 180,E1 -15021.312,E2 -15021.312} C_VEL
LIN {X 0,Y 325.241,Z 605.617,A -85,B 0,C 180,E1 -15023.798,E2 -15023.798} C_VEL
LIN {X 0,Y 325.008,Z 607.919,A -85,B 0,C 180,E1 -15026.281,E2 -15026.281} C_VEL
LIN {X 0,Y 324.868,Z 609.095,A -85,B 0,C 180,E1 -15028.76,E2 -15028.76} C_VEL
LIN {X 0,Y 324.868,Z 609.109,A -85,B 0,C 180,E1 -15031.24,E2 -15031.24} C_VEL
LIN {X 0,Y 325.003,Z 607.991,A -85,B 0,C 180,E1 -15033.719,E2 -15033.719} C_VEL
LIN {X 0,Y 325.231,Z 605.672,A -85,B 0,C 180,E1 -15036.265,E2 -15036.265} C_VEL
LIN {X 0,Y 325.637,Z 602.313,A -85,B 0,C 180,E1 -15038.689,E2 -15038.689} C_VEL
LIN {X 0,Y 326.33,Z 597.614,A -85,B 0,C 180,E1 -15041.176,E2 -15041.176} C_VEL
LIN {X 0,Y 327.452,Z 591.519,A -85,B 0,C 180,E1 -15043.655,E2 -15043.655} C_VEL
LIN {X 0,Y 328.83,Z 583.845,A -85,B 0,C 180,E1 -15046.131,E2 -15046.131} C_VEL
LIN {X 0,Y 330.494,Z 575.656,A -85,B 0,C 180,E1 -15048.279,E2 -15048.279} C_VEL
LIN {X 0,Y 332.467,Z 565.789,A -85,B 0,C 180,E1 -15050.413,E2 -15050.413} C_VEL
LIN {X 0,Y 334.447,Z 555.669,A -85,B 0,C 180,E1 -15052.225,E2 -15052.225} C_VEL
LIN {X 0,Y 336.727,Z 543.613,A -85,B 0,C 180,E1 -15054.015,E2 -15054.015} C_VEL
LIN {X 0,Y 338.89,Z 531.52,A -85,B 0,C 180,E1 -15055.487,E2 -15055.487} C_VEL
LIN {X 0,Y 340.956,Z 518.376,A -85,B 0,C 180,E1 -15056.801,E2 -15056.801} C_VEL
LIN {X 0,Y 342.628,Z 505.846,A -85,B 0,C 180,E1 -15057.816,E2 -15057.816} C_VEL
LIN {X 0,Y 344.179,Z 491.047,A -85,B 0,C 180,E1 -15058.767,E2 -15058.767} C_VEL
LIN {X 0,Y 345.435,Z 475.921,A -85,B 0,C 180,E1 -15059.478,E2 -15059.478} C_VEL
LIN {X 0,Y 346.381,Z 461.208,A -85,B 0,C 180,E1 -15059.933,E2 -15059.933} C_VEL
LIN {X 0,Y 346.478,Z 458.824,A -85,B 0,C 180,E1 -15059.99,E2 -15059.99} C_VEL
LIN {X 0,Y 346.093,Z 453.039,A -85,B 0,C 180,E1 -15060.181,E2 -15060.181} C_VEL
LIN {X 0,Y 341.696,Z 434.42,A -85,B 0,C 180,E1 -15061.055,E2 -15061.055} C_VEL
LIN {X 0,Y 341.337,Z 428.619,A -85,B 0,C 180,E1 -15061.228,E2 -15061.228} C_VEL
LIN {X 0,Y 343.888,Z 347.353,A -85,B 0,C 180,E1 -15062.932,E2 -15062.932} C_VEL
LIN {X 0,Y 335.896,Z 329.746,A -85,B 0,C 180,E1 -15064.272,E2 -15064.272} C_VEL
LIN {X 0,Y 326.114,Z 310.995,A -85,B 0,C 180,E1 -15065.958,E2 -15065.958} C_VEL
LIN {X 0,Y 321.414,Z 302.781,A -85,B 0,C 180,E1 -15066.797,E2 -15066.797} C_VEL
LIN {X 0,Y 320.08,Z 300.163,A -85,B 0,C 180,E1 -15067.078,E2 -15067.078} C_VEL
LIN {X 0,Y 319.569,Z 298.302,A -85,B 0,C 180,E1 -15067.719,E2 -15067.719} C_VEL
LIN {X 0,Y 319.522,Z 298.308,A -85,B 0,C 180,E1 -15071.596,E2 -15071.596} C_VEL
LIN {X 0,Y 319.484,Z 298.313,A -85,B 0,C 180,E1 -15075.256,E2 -15075.256} C_VEL
LIN {X 0,Y 319.522,Z 298.292,A -85,B 0,C 180,E1 -15078.711,E2 -15078.711} C_VEL
LIN {X 0,Y 319.547,Z 298.29,A -85,B 0,C 180,E1 -15082.349,E2 -15082.349} C_VEL
LIN {X 0,Y 319.552,Z 298.298,A -85,B 0,C 180,E1 -15085.122,E2 -15085.122} C_VEL
LIN {X 0,Y 319.517,Z 298.292,A -85,B 0,C 180,E1 -15088.136,E2 -15088.136} C_VEL
LIN {X 0,Y 319.597,Z 298.295,A -85,B 0,C 180,E1 -15091.592,E2 -15091.592} C_VEL
LIN {X 0,Y 319.578,Z 298.299,A -85,B 0,C 180,E1 -15095.302,E2 -15095.302} C_VEL
LIN {X 0,Y 319.558,Z 298.297,A -85,B 0,C 180,E1 -15098.045,E2 -15098.045} C_VEL
LIN {X 0,Y 319.616,Z 298.289,A -85,B 0,C 180,E1 -15102.07,E2 -15102.07} C_VEL
LIN {X 0,Y 319.722,Z 298.278,A -85,B 0,C 180,E1 -15106.007,E2 -15106.007} C_VEL
LIN {X 0,Y 319.726,Z 298.28,A -85,B 0,C 180,E1 -15109.872,E2 -15109.872} C_VEL
LIN {X 0,Y 319.905,Z 298.26,A -85,B 0,C 180,E1 -15113.693,E2 -15113.693} C_VEL
LIN {X 0,Y 319.966,Z 298.253,A -85,B 0,C 180,E1 -15117.482,E2 -15117.482} C_VEL
LIN {X 0,Y 320.085,Z 298.229,A -85,B 0,C 180,E1 -15120,E2 -15120} C_VEL
LIN {X 0,Y 319.947,Z 298.258,A -85,B 0,C 180,E1 -15122.518,E2 -15122.518} C_VEL
LIN {X 0,Y 319.899,Z 298.261,A -85,B 0,C 180,E1 -15126.306,E2 -15126.306} C_VEL
LIN {X 0,Y 319.725,Z 298.278,A -85,B 0,C 180,E1 -15130.128,E2 -15130.128} C_VEL
LIN {X 0,Y 319.721,Z 298.276,A -85,B 0,C 180,E1 -15133.993,E2 -15133.993} C_VEL
LIN {X 0,Y 319.605,Z 298.292,A -85,B 0,C 180,E1 -15137.93,E2 -15137.93} C_VEL
LIN {X 0,Y 319.556,Z 298.299,A -85,B 0,C 180,E1 -15141.955,E2 -15141.955} C_VEL
LIN {X 0,Y 319.544,Z 298.3,A -85,B 0,C 180,E1 -15146.096,E2 -15146.096} C_VEL
LIN {X 0,Y 319.535,Z 298.308,A -85,B 0,C 180,E1 -15148.939,E2 -15148.939} C_VEL
LIN {X 0,Y 319.516,Z 298.311,A -85,B 0,C 180,E1 -15151.863,E2 -15151.863} C_VEL
LIN {X 0,Y 319.57,Z 298.301,A -85,B 0,C 180,E1 -15155.543,E2 -15155.543} C_VEL
LIN {X 0,Y 319.525,Z 298.31,A -85,B 0,C 180,E1 -15158.015,E2 -15158.015} C_VEL
LIN {X 0,Y 319.498,Z 298.293,A -85,B 0,C 180,E1 -15161.593,E2 -15161.593} C_VEL
LIN {X 0,Y 319.48,Z 298.313,A -85,B 0,C 180,E1 -15164.744,E2 -15164.744} C_VEL
LIN {X 0,Y 319.544,Z 298.306,A -85,B 0,C 180,E1 -15167.016,E2 -15167.016} C_VEL
LIN {X 0,Y 319.504,Z 298.398,A -85,B 0,C 180,E1 -15168.709,E2 -15168.709} C_VEL
LIN {X 0,Y 322.868,Z 309.683,A -85,B 0,C 180,E1 -15172.122,E2 -15172.122} C_VEL
LIN {X 0,Y 324.317,Z 314.875,A -85,B 0,C 180,E1 -15173.557,E2 -15173.557} C_VEL
LIN {X 0,Y 333.231,Z 332.726,A -85,B 0,C 180,E1 -15175.133,E2 -15175.133} C_VEL
LIN {X 0,Y 340.475,Z 348.959,A -85,B 0,C 180,E1 -15176.375,E2 -15176.375} C_VEL
LIN {X 0,Y 343.368,Z 365.505,A -85,B 0,C 180,E1 -15177.097,E2 -15177.097} C_VEL
LIN {X 0,Y 340.484,Z 459.151,A -85,B 0,C 180,E1 -15179.064,E2 -15179.064} C_VEL
LIN {X 0,Y 339.553,Z 483.46,A -85,B 0,C 180,E1 -15179.616,E2 -15179.616} C_VEL
LIN {X 0,Y 338.386,Z 498.108,A -85,B 0,C 180,E1 -15180.146,E2 -15180.146} C_VEL
LIN {X 0,Y 336.803,Z 512.635,A -85,B 0,C 180,E1 -15180.893,E2 -15180.893} C_VEL
LIN {X 0,Y 334.859,Z 527.266,A -85,B 0,C 180,E1 -15181.903,E2 -15181.903} C_VEL
LIN {X 0,Y 332.659,Z 541.385,A -85,B 0,C 180,E1 -15183.155,E2 -15183.155} C_VEL
LIN {X 0,Y 330.274,Z 554.819,A -85,B 0,C 180,E1 -15184.644,E2 -15184.644} C_VEL
LIN {X 0,Y 327.866,Z 567.058,A -85,B 0,C 180,E1 -15186.303,E2 -15186.303} C_VEL
LIN {X 0,Y 325.613,Z 578.24,A -85,B 0,C 180,E1 -15188.142,E2 -15188.142} C_VEL
LIN {X 0,Y 323.766,Z 587.656,A -85,B 0,C 180,E1 -15190.009,E2 -15190.009} C_VEL
LIN {X 0,Y 321.827,Z 596.921,A -85,B 0,C 180,E1 -15192.198,E2 -15192.198} C_VEL
LIN {X 0,Y 320.197,Z 605.65,A -85,B 0,C 180,E1 -15194.729,E2 -15194.729} C_VEL
LIN {X 0,Y 319.097,Z 612.662,A -85,B 0,C 180,E1 -15197.277,E2 -15197.277} C_VEL
LIN {X 0,Y 318.292,Z 618.177,A -85,B 0,C 180,E1 -15199.826,E2 -15199.826} C_VEL
LIN {X 0,Y 317.917,Z 622.352,A -85,B 0,C 180,E1 -15202.378,E2 -15202.378} C_VEL
LIN {X 0,Y 317.774,Z 625.282,A -85,B 0,C 180,E1 -15204.925,E2 -15204.925} C_VEL
LIN {X 0,Y 317.746,Z 627.029,A -85,B 0,C 180,E1 -15207.465,E2 -15207.465} C_VEL
LIN {X 0,Y 317.78,Z 627.627,A -85,B 0,C 180,E1 -15210,E2 -15210} C_VEL
LIN {X 0,Y 317.745,Z 627.02,A -85,B 0,C 180,E1 -15212.535,E2 -15212.535} C_VEL
LIN {X 0,Y 317.764,Z 625.261,A -85,B 0,C 180,E1 -15215.075,E2 -15215.075} C_VEL
LIN {X 0,Y 317.914,Z 622.326,A -85,B 0,C 180,E1 -15217.622,E2 -15217.622} C_VEL
LIN {X 0,Y 318.291,Z 618.147,A -85,B 0,C 180,E1 -15220.174,E2 -15220.174} C_VEL
LIN {X 0,Y 319.093,Z 612.618,A -85,B 0,C 180,E1 -15222.723,E2 -15222.723} C_VEL
LIN {X 0,Y 320.168,Z 605.586,A -85,B 0,C 180,E1 -15225.272,E2 -15225.272} C_VEL
LIN {X 0,Y 321.855,Z 596.847,A -85,B 0,C 180,E1 -15227.8,E2 -15227.8} C_VEL
LIN {X 0,Y 323.469,Z 589.018,A -85,B 0,C 180,E1 -15229.679,E2 -15229.679} C_VEL
LIN {X 0,Y 325.308,Z 579.781,A -85,B 0,C 180,E1 -15231.547,E2 -15231.547} C_VEL
LIN {X 0,Y 327.453,Z 568.904,A -85,B 0,C 180,E1 -15233.394,E2 -15233.394} C_VEL
LIN {X 0,Y 329.799,Z 557.04,A -85,B 0,C 180,E1 -15235.057,E2 -15235.057} C_VEL
LIN {X 0,Y 332.197,Z 544.069,A -85,B 0,C 180,E1 -15236.546,E2 -15236.546} C_VEL
LIN {X 0,Y 334.434,Z 530.137,A -85,B 0,C 180,E1 -15237.838,E2 -15237.838} C_VEL
LIN {X 0,Y 336.384,Z 515.75,A -85,B 0,C 180,E1 -15238.89,E2 -15238.89} C_VEL
LIN {X 0,Y 338.036,Z 500.788,A -85,B 0,C 180,E1 -15239.717,E2 -15239.717} C_VEL
LIN {X 0,Y 339.324,Z 485.163,A -85,B 0,C 180,E1 -15240.32,E2 -15240.32} C_VEL
LIN {X 0,Y 340.213,Z 465.389,A -85,B 0,C 180,E1 -15240.791,E2 -15240.791} C_VEL
LIN {X 0,Y 343.327,Z 365.376,A -85,B 0,C 180,E1 -15242.887,E2 -15242.887} C_VEL
LIN {X 0,Y 340.238,Z 348.339,A -85,B 0,C 180,E1 -15243.642,E2 -15243.642} C_VEL
LIN {X 0,Y 332.281,Z 330.741,A -85,B 0,C 180,E1 -15245.005,E2 -15245.005} C_VEL
LIN {X 0,Y 324.221,Z 314.508,A -85,B 0,C 180,E1 -15246.463,E2 -15246.463} C_VEL
LIN {X 0,Y 320.8,Z 302.666,A -85,B 0,C 180,E1 -15249.935,E2 -15249.935} C_VEL
LIN {X 0,Y 319.493,Z 298.313,A -85,B 0,C 180,E1 -15251.292,E2 -15251.292} C_VEL
LIN {X 0,Y 319.514,Z 298.311,A -85,B 0,C 180,E1 -15253.459,E2 -15253.459} C_VEL
LIN {X 0,Y 319.545,Z 298.305,A -85,B 0,C 180,E1 -15257.015,E2 -15257.015} C_VEL
LIN {X 0,Y 319.508,Z 298.312,A -85,B 0,C 180,E1 -15260.365,E2 -15260.365} C_VEL
LIN {X 0,Y 319.547,Z 298.306,A -85,B 0,C 180,E1 -15263.571,E2 -15263.571} C_VEL
LIN {X 0,Y 319.57,Z 298.298,A -85,B 0,C 180,E1 -15266.686,E2 -15266.686} C_VEL
LIN {X 0,Y 319.552,Z 298.301,A -85,B 0,C 180,E1 -15269.613,E2 -15269.613} C_VEL
LIN {X 0,Y 319.53,Z 298.303,A -85,B 0,C 180,E1 -15272.491,E2 -15272.491} C_VEL
LIN {X 0,Y 319.519,Z 298.308,A -85,B 0,C 180,E1 -15275.297,E2 -15275.297} C_VEL
LIN {X 0,Y 319.556,Z 298.304,A -85,B 0,C 180,E1 -15278.045,E2 -15278.045} C_VEL
LIN {X 0,Y 319.605,Z 298.276,A -85,B 0,C 180,E1 -15282.07,E2 -15282.07} C_VEL
LIN {X 0,Y 319.721,Z 298.277,A -85,B 0,C 180,E1 -15286.007,E2 -15286.007} C_VEL
LIN {X 0,Y 319.723,Z 298.26,A -85,B 0,C 180,E1 -15289.872,E2 -15289.872} C_VEL
LIN {X 0,Y 319.894,Z 298.256,A -85,B 0,C 180,E1 -15293.694,E2 -15293.694} C_VEL
LIN {X 0,Y 319.946,Z 298.252,A -85,B 0,C 180,E1 -15297.482,E2 -15297.482} C_VEL
LIN {X 0,Y 319.988,Z 298.251,A -85,B 0,C 180,E1 -15301.259,E2 -15301.259} C_VEL
LIN {X 0,Y 319.704,Z 298.285,A -85,B 0,C 180,E1 -15303.781,E2 -15303.781} C_VEL
LIN {X 0,Y 319.881,Z 298.257,A -85,B 0,C 180,E1 -15306.565,E2 -15306.565} C_VEL
LIN {X 0,Y 319.726,Z 298.279,A -85,B 0,C 180,E1 -15310.128,E2 -15310.128} C_VEL
LIN {X 0,Y 319.722,Z 298.28,A -85,B 0,C 180,E1 -15313.993,E2 -15313.993} C_VEL
LIN {X 0,Y 319.605,Z 298.294,A -85,B 0,C 180,E1 -15317.93,E2 -15317.93} C_VEL
LIN {X 0,Y 319.56,Z 298.286,A -85,B 0,C 180,E1 -15321.955,E2 -15321.955} C_VEL
LIN {X 0,Y 319.586,Z 298.287,A -85,B 0,C 180,E1 -15326.093,E2 -15326.093} C_VEL
LIN {X 0,Y 319.57,Z 298.29,A -85,B 0,C 180,E1 -15328.936,E2 -15328.936} C_VEL
LIN {X 0,Y 319.524,Z 298.303,A -85,B 0,C 180,E1 -15331.863,E2 -15331.863} C_VEL
LIN {X 0,Y 319.572,Z 298.301,A -85,B 0,C 180,E1 -15335.543,E2 -15335.543} C_VEL
LIN {X 0,Y 319.554,Z 298.301,A -85,B 0,C 180,E1 -15339.67,E2 -15339.67} C_VEL
LIN {X 0,Y 319.517,Z 298.31,A -85,B 0,C 180,E1 -15343.461,E2 -15343.461} C_VEL
LIN {X 0,Y 319.55,Z 298.305,A -85,B 0,C 180,E1 -15347.017,E2 -15347.017} C_VEL
LIN {X 0,Y 319.544,Z 298.301,A -85,B 0,C 180,E1 -15350.372,E2 -15350.372} C_VEL
LIN {X 0,Y 319.572,Z 298.362,A -85,B 0,C 180,E1 -15352.456,E2 -15352.456} C_VEL
LIN {X 0,Y 320.274,Z 300.551,A -85,B 0,C 180,E1 -15353.109,E2 -15353.109} C_VEL
LIN {X 0,Y 322.36,Z 304.242,A -85,B 0,C 180,E1 -15353.49,E2 -15353.49} C_VEL
LIN {X 0,Y 331.882,Z 321.808,A -85,B 0,C 180,E1 -15355.163,E2 -15355.163} C_VEL
LIN {X 0,Y 340.646,Z 339.974,A -85,B 0,C 180,E1 -15356.643,E2 -15356.643} C_VEL
LIN {X 0,Y 343.81,Z 347.136,A -85,B 0,C 180,E1 -15357.168,E2 -15357.168} C_VEL
LIN {X 0,Y 340.908,Z 439.641,A -85,B 0,C 180,E1 -15359.107,E2 -15359.107} C_VEL
LIN {X 0,Y 339.88,Z 466.061,A -85,B 0,C 180,E1 -15359.692,E2 -15359.692} C_VEL
LIN {X 0,Y 338.827,Z 481.579,A -85,B 0,C 180,E1 -15360.27,E2 -15360.27} C_VEL
LIN {X 0,Y 337.571,Z 495.014,A -85,B 0,C 180,E1 -15360.976,E2 -15360.976} C_VEL
LIN {X 0,Y 336.007,Z 508.694,A -85,B 0,C 180,E1 -15361.927,E2 -15361.927} C_VEL
LIN {X 0,Y 333.933,Z 522.261,A -85,B 0,C 180,E1 -15363.097,E2 -15363.097} C_VEL
LIN {X 0,Y 331.898,Z 534.734,A -85,B 0,C 180,E1 -15364.442,E2 -15364.442} C_VEL
LIN {X 0,Y 329.68,Z 546.308,A -85,B 0,C 180,E1 -15365.94,E2 -15365.94} C_VEL
LIN {X 0,Y 328.01,Z 555.276,A -85,B 0,C 180,E1 -15367.315,E2 -15367.315} C_VEL
LIN {X 0,Y 325.881,Z 565.457,A -85,B 0,C 180,E1 -15369.156,E2 -15369.156} C_VEL
LIN {X 0,Y 323.806,Z 575.413,A -85,B 0,C 180,E1 -15371.329,E2 -15371.329} C_VEL
LIN {X 0,Y 321.993,Z 583.67,A -85,B 0,C 180,E1 -15373.517,E2 -15373.517} C_VEL
LIN {X 0,Y 320.546,Z 591.416,A -85,B 0,C 180,E1 -15376.044,E2 -15376.044} C_VEL
LIN {X 0,Y 319.358,Z 597.582,A -85,B 0,C 180,E1 -15378.577,E2 -15378.577} C_VEL
LIN {X 0,Y 318.636,Z 602.338,A -85,B 0,C 180,E1 -15381.119,E2 -15381.119} C_VEL
LIN {X 0,Y 318.16,Z 605.908,A -85,B 0,C 180,E1 -15383.736,E2 -15383.736} C_VEL
LIN {X 0,Y 317.94,Z 608.122,A -85,B 0,C 180,E1 -15386.198,E2 -15386.198} C_VEL
LIN {X 0,Y 317.779,Z 609.298,A -85,B 0,C 180,E1 -15388.733,E2 -15388.733} C_VEL
LIN {X 0,Y 317.778,Z 609.312,A -85,B 0,C 180,E1 -15391.267,E2 -15391.267} C_VEL
LIN {X 0,Y 317.935,Z 608.193,A -85,B 0,C 180,E1 -15393.802,E2 -15393.802} C_VEL
LIN {X 0,Y 318.166,Z 605.947,A -85,B 0,C 180,E1 -15396.341,E2 -15396.341} C_VEL
LIN {X 0,Y 318.611,Z 602.516,A -85,B 0,C 180,E1 -15398.882,E2 -15398.882} C_VEL
LIN {X 0,Y 319.329,Z 597.816,A -85,B 0,C 180,E1 -15401.424,E2 -15401.424} C_VEL
LIN {X 0,Y 320.515,Z 591.721,A -85,B 0,C 180,E1 -15403.957,E2 -15403.957} C_VEL
LIN {X 0,Y 321.984,Z 584.047,A -85,B 0,C 180,E1 -15406.484,E2 -15406.484} C_VEL
LIN {X 0,Y 323.728,Z 575.858,A -85,B 0,C 180,E1 -15408.675,E2 -15408.675} C_VEL
LIN {X 0,Y 325.796,Z 565.99,A -85,B 0,C 180,E1 -15410.85,E2 -15410.85} C_VEL
LIN {X 0,Y 327.849,Z 555.87,A -85,B 0,C 180,E1 -15412.696,E2 -15412.696} C_VEL
LIN {X 0,Y 330.229,Z 543.813,A -85,B 0,C 180,E1 -15414.519,E2 -15414.519} C_VEL
LIN {X 0,Y 332.467,Z 531.719,A -85,B 0,C 180,E1 -15416.016,E2 -15416.016} C_VEL
LIN {X 0,Y 334.614,Z 518.574,A -85,B 0,C 180,E1 -15417.351,E2 -15417.351} C_VEL
LIN {X 0,Y 336.366,Z 506.043,A -85,B 0,C 180,E1 -15418.38,E2 -15418.38} C_VEL
LIN {X 0,Y 338.005,Z 490.853,A -85,B 0,C 180,E1 -15419.369,E2 -15419.369} C_VEL
LIN {X 0,Y 339.281,Z 476.112,A -85,B 0,C 180,E1 -15420.067,E2 -15420.067} C_VEL
LIN {X 0,Y 340.26,Z 461.39,A -85,B 0,C 180,E1 -15420.528,E2 -15420.528} C_VEL
LIN {X 0,Y 341.337,Z 428.619,A -85,B 0,C 180,E1 -15421.228,E2 -15421.228} C_VEL
LIN {X 0,Y 340.983,Z 422.82,A -85,B 0,C 180,E1 -15421.405,E2 -15421.405} C_VEL
LIN {X 0,Y 336.696,Z 404.21,A -85,B 0,C 180,E1 -15422.314,E2 -15422.314} C_VEL
LIN {X 0,Y 336.331,Z 398.411,A -85,B 0,C 180,E1 -15422.498,E2 -15422.498} C_VEL
LIN {X 0,Y 337.885,Z 349.389,A -85,B 0,C 180,E1 -15423.548,E2 -15423.548} C_VEL
LIN {X 0,Y 329.799,Z 331.685,A -85,B 0,C 180,E1 -15424.951,E2 -15424.951} C_VEL
LIN {X 0,Y 320.099,Z 313.045,A -85,B 0,C 180,E1 -15426.692,E2 -15426.692} C_VEL
LIN {X 0,Y 313.706,Z 302.32,A -85,B 0,C 180,E1 -15427.878,E2 -15427.878} C_VEL
LIN {X 0,Y 312.808,Z 300.482,A -85,B 0,C 180,E1 -15428.072,E2 -15428.072} C_VEL
LIN {X 0,Y 312.501,Z 299.189,A -85,B 0,C 180,E1 -15428.5,E2 -15428.5} C_VEL
LIN {X 0,Y 312.486,Z 299.188,A -85,B 0,C 180,E1 -15432.431,E2 -15432.431} C_VEL
LIN {X 0,Y 312.454,Z 299.19,A -85,B 0,C 180,E1 -15436.034,E2 -15436.034} C_VEL
LIN {X 0,Y 312.499,Z 299.18,A -85,B 0,C 180,E1 -15439.874,E2 -15439.874} C_VEL
LIN {X 0,Y 312.528,Z 299.161,A -85,B 0,C 180,E1 -15444.05,E2 -15444.05} C_VEL
LIN {X 0,Y 312.495,Z 299.176,A -85,B 0,C 180,E1 -15447.333,E2 -15447.333} C_VEL
LIN {X 0,Y 312.526,Z 299.17,A -85,B 0,C 180,E1 -15451.282,E2 -15451.282} C_VEL
LIN {X 0,Y 312.551,Z 299.171,A -85,B 0,C 180,E1 -15454.708,E2 -15454.708} C_VEL
LIN {X 0,Y 312.519,Z 299.175,A -85,B 0,C 180,E1 -15458.911,E2 -15458.911} C_VEL
LIN {X 0,Y 312.574,Z 299.168,A -85,B 0,C 180,E1 -15461.652,E2 -15461.652} C_VEL
LIN {X 0,Y 312.676,Z 299.156,A -85,B 0,C 180,E1 -15465.685,E2 -15465.685} C_VEL
LIN {X 0,Y 312.676,Z 299.159,A -85,B 0,C 180,E1 -15469.641,E2 -15469.641} C_VEL
LIN {X 0,Y 312.819,Z 299.139,A -85,B 0,C 180,E1 -15472.253,E2 -15472.253} C_VEL
LIN {X 0,Y 312.69,Z 299.152,A -85,B 0,C 180,E1 -15474.842,E2 -15474.842} C_VEL
LIN {X 0,Y 312.973,Z 299.122,A -85,B 0,C 180,E1 -15478.713,E2 -15478.713} C_VEL
LIN {X 0,Y 312.971,Z 299.122,A -85,B 0,C 180,E1 -15481.287,E2 -15481.287} C_VEL
LIN {X 0,Y 312.842,Z 299.141,A -85,B 0,C 180,E1 -15486.449,E2 -15486.449} C_VEL
LIN {X 0,Y 312.741,Z 299.145,A -85,B 0,C 180,E1 -15489.05,E2 -15489.05} C_VEL
LIN {X 0,Y 312.622,Z 299.161,A -85,B 0,C 180,E1 -15492.991,E2 -15492.991} C_VEL
LIN {X 0,Y 312.613,Z 299.171,A -85,B 0,C 180,E1 -15495.651,E2 -15495.651} C_VEL
LIN {X 0,Y 312.529,Z 299.182,A -85,B 0,C 180,E1 -15499.713,E2 -15499.713} C_VEL
LIN {X 0,Y 312.508,Z 299.18,A -85,B 0,C 180,E1 -15502.776,E2 -15502.776} C_VEL
LIN {X 0,Y 312.478,Z 299.183,A -85,B 0,C 180,E1 -15506.732,E2 -15506.732} C_VEL
LIN {X 0,Y 312.488,Z 299.186,A -85,B 0,C 180,E1 -15509.656,E2 -15509.656} C_VEL
LIN {X 0,Y 312.512,Z 299.175,A -85,B 0,C 180,E1 -15513.689,E2 -15513.689} C_VEL
LIN {X 0,Y 312.506,Z 299.181,A -85,B 0,C 180,E1 -15517.388,E2 -15517.388} C_VEL
LIN {X 0,Y 312.434,Z 299.167,A -85,B 0,C 180,E1 -15520.718,E2 -15520.718} C_VEL
LIN {X 0,Y 312.444,Z 299.188,A -85,B 0,C 180,E1 -15524.211,E2 -15524.211} C_VEL
LIN {X 0,Y 312.458,Z 299.201,A -85,B 0,C 180,E1 -15527.857,E2 -15527.857} C_VEL
LIN {X 0,Y 315.663,Z 309.793,A -85,B 0,C 180,E1 -15531.192,E2 -15531.192} C_VEL
LIN {X 0,Y 316.969,Z 314.481,A -85,B 0,C 180,E1 -15532.565,E2 -15532.565} C_VEL
LIN {X 0,Y 326.127,Z 332.399,A -85,B 0,C 180,E1 -15534.256,E2 -15534.256} C_VEL
LIN {X 0,Y 334.506,Z 350.965,A -85,B 0,C 180,E1 -15535.748,E2 -15535.748} C_VEL
LIN {X 0,Y 335.56,Z 355.511,A -85,B 0,C 180,E1 -15535.985,E2 -15535.985} C_VEL
LIN {X 0,Y 337.416,Z 367.202,A -85,B 0,C 180,E1 -15536.488,E2 -15536.488} C_VEL
LIN {X 0,Y 333.831,Z 474.868,A -85,B 0,C 180,E1 -15538.775,E2 -15538.775} C_VEL
LIN {X 0,Y 332.905,Z 489.904,A -85,B 0,C 180,E1 -15539.207,E2 -15539.207} C_VEL
LIN {X 0,Y 331.529,Z 504.713,A -85,B 0,C 180,E1 -15539.859,E2 -15539.859} C_VEL
LIN {X 0,Y 329.682,Z 519.647,A -85,B 0,C 180,E1 -15540.765,E2 -15540.765} C_VEL
LIN {X 0,Y 327.673,Z 533.307,A -85,B 0,C 180,E1 -15541.846,E2 -15541.846} C_VEL
LIN {X 0,Y 325.281,Z 546.9,A -85,B 0,C 180,E1 -15543.191,E2 -15543.191} C_VEL
LIN {X 0,Y 322.638,Z 560.471,A -85,B 0,C 180,E1 -15544.865,E2 -15544.865} C_VEL
LIN {X 0,Y 320.116,Z 572.687,A -85,B 0,C 180,E1 -15546.723,E2 -15546.723} C_VEL
LIN {X 0,Y 318.026,Z 582.949,A -85,B 0,C 180,E1 -15548.616,E2 -15548.616} C_VEL
LIN {X 0,Y 315.762,Z 592.977,A -85,B 0,C 180,E1 -15550.835,E2 -15550.835} C_VEL
LIN {X 0,Y 314.057,Z 601.313,A -85,B 0,C 180,E1 -15553.088,E2 -15553.088} C_VEL
LIN {X 0,Y 312.628,Z 609.151,A -85,B 0,C 180,E1 -15555.684,E2 -15555.684} C_VEL
LIN {X 0,Y 311.604,Z 615.391,A -85,B 0,C 180,E1 -15558.289,E2 -15558.289} C_VEL
LIN {X 0,Y 311.008,Z 620.222,A -85,B 0,C 180,E1 -15560.899,E2 -15560.899} C_VEL
LIN {X 0,Y 310.778,Z 623.766,A -85,B 0,C 180,E1 -15563.508,E2 -15563.508} C_VEL
LIN {X 0,Y 310.676,Z 626.097,A -85,B 0,C 180,E1 -15566.109,E2 -15566.109} C_VEL
LIN {X 0,Y 310.653,Z 627.269,A -85,B 0,C 180,E1 -15568.704,E2 -15568.704} C_VEL
LIN {X 0,Y 310.653,Z 627.266,A -85,B 0,C 180,E1 -15571.296,E2 -15571.296} C_VEL
LIN {X 0,Y 310.672,Z 626.082,A -85,B 0,C 180,E1 -15573.891,E2 -15573.891} C_VEL
LIN {X 0,Y 310.712,Z 623.739,A -85,B 0,C 180,E1 -15576.494,E2 -15576.494} C_VEL
LIN {X 0,Y 311.003,Z 620.192,A -85,B 0,C 180,E1 -15579.101,E2 -15579.101} C_VEL
LIN {X 0,Y 311.603,Z 615.353,A -85,B 0,C 180,E1 -15581.711,E2 -15581.711} C_VEL
LIN {X 0,Y 312.605,Z 609.094,A -85,B 0,C 180,E1 -15584.318,E2 -15584.318} C_VEL
LIN {X 0,Y 314.062,Z 601.24,A -85,B 0,C 180,E1 -15586.912,E2 -15586.912} C_VEL
LIN {X 0,Y 315.771,Z 592.894,A -85,B 0,C 180,E1 -15589.164,E2 -15589.164} C_VEL
LIN {X 0,Y 318.044,Z 582.85,A -85,B 0,C 180,E1 -15591.383,E2 -15591.383} C_VEL
LIN {X 0,Y 320.128,Z 572.577,A -85,B 0,C 180,E1 -15593.276,E2 -15593.276} C_VEL
LIN {X 0,Y 322.433,Z 561.418,A -85,B 0,C 180,E1 -15594.98,E2 -15594.98} C_VEL
LIN {X 0,Y 324.755,Z 549.361,A -85,B 0,C 180,E1 -15596.509,E2 -15596.509} C_VEL
LIN {X 0,Y 327.097,Z 536.293,A -85,B 0,C 180,E1 -15597.86,E2 -15597.86} C_VEL
LIN {X 0,Y 329.2,Z 522.563,A -85,B 0,C 180,E1 -15599.002,E2 -15599.002} C_VEL
LIN {X 0,Y 331.033,Z 508.29,A -85,B 0,C 180,E1 -15599.927,E2 -15599.927} C_VEL
LIN {X 0,Y 332.613,Z 493.095,A -85,B 0,C 180,E1 -15600.646,E2 -15600.646} C_VEL
LIN {X 0,Y 333.625,Z 478.58,A -85,B 0,C 180,E1 -15601.114,E2 -15601.114} C_VEL
LIN {X 0,Y 337.379,Z 367.156,A -85,B 0,C 180,E1 -15603.493,E2 -15603.493} C_VEL
LIN {X 0,Y 334.583,Z 351.16,A -85,B 0,C 180,E1 -15604.212,E2 -15604.212} C_VEL
LIN {X 0,Y 327.084,Z 334.448,A -85,B 0,C 180,E1 -15605.542,E2 -15605.542} C_VEL
LIN {X 0,Y 318.99,Z 318.371,A -85,B 0,C 180,E1 -15607.02,E2 -15607.02} C_VEL
LIN {X 0,Y 316.923,Z 314.329,A -85,B 0,C 180,E1 -15607.424,E2 -15607.424} C_VEL
LIN {X 0,Y 313.56,Z 302.951,A -85,B 0,C 180,E1 -15610.905,E2 -15610.905} C_VEL
LIN {X 0,Y 312.465,Z 299.192,A -85,B 0,C 180,E1 -15612.142,E2 -15612.142} C_VEL
LIN {X 0,Y 312.451,Z 299.193,A -85,B 0,C 180,E1 -15616.035,E2 -15616.035} C_VEL
LIN {X 0,Y 312.448,Z 299.188,A -85,B 0,C 180,E1 -15619.885,E2 -15619.885} C_VEL
LIN {X 0,Y 312.525,Z 299.176,A -85,B 0,C 180,E1 -15624.051,E2 -15624.051} C_VEL
LIN {X 0,Y 312.494,Z 299.178,A -85,B 0,C 180,E1 -15627.333,E2 -15627.333} C_VEL
LIN {X 0,Y 312.498,Z 299.183,A -85,B 0,C 180,E1 -15631.292,E2 -15631.292} C_VEL
LIN {X 0,Y 312.509,Z 299.182,A -85,B 0,C 180,E1 -15634.704,E2 -15634.704} C_VEL
LIN {X 0,Y 312.531,Z 299.181,A -85,B 0,C 180,E1 -15637.525,E2 -15637.525} C_VEL
LIN {X 0,Y 312.558,Z 299.149,A -85,B 0,C 180,E1 -15641.652,E2 -15641.652} C_VEL
LIN {X 0,Y 312.676,Z 299.157,A -85,B 0,C 180,E1 -15645.686,E2 -15645.686} C_VEL
LIN {X 0,Y 312.673,Z 299.133,A -85,B 0,C 180,E1 -15649.641,E2 -15649.641} C_VEL
LIN {X 0,Y 312.835,Z 299.136,A -85,B 0,C 180,E1 -15653.551,E2 -15653.551} C_VEL
LIN {X 0,Y 312.971,Z 299.116,A -85,B 0,C 180,E1 -15658.713,E2 -15658.713} C_VEL
LIN {X 0,Y 312.899,Z 299.125,A -85,B 0,C 180,E1 -15662.575,E2 -15662.575} C_VEL
LIN {X 0,Y 312.835,Z 299.135,A -85,B 0,C 180,E1 -15666.547,E2 -15666.547} C_VEL
LIN {X 0,Y 312.742,Z 299.155,A -85,B 0,C 180,E1 -15669.051,E2 -15669.051} C_VEL
LIN {X 0,Y 312.623,Z 299.17,A -85,B 0,C 180,E1 -15672.992,E2 -15672.992} C_VEL
LIN {X 0,Y 312.613,Z 299.166,A -85,B 0,C 180,E1 -15675.651,E2 -15675.651} C_VEL
LIN {X 0,Y 312.531,Z 299.153,A -85,B 0,C 180,E1 -15679.713,E2 -15679.713} C_VEL
LIN {X 0,Y 312.518,Z 299.173,A -85,B 0,C 180,E1 -15682.781,E2 -15682.781} C_VEL
LIN {X 0,Y 312.563,Z 299.164,A -85,B 0,C 180,E1 -15685.924,E2 -15685.924} C_VEL
LIN {X 0,Y 312.53,Z 299.177,A -85,B 0,C 180,E1 -15689.652,E2 -15689.652} C_VEL
LIN {X 0,Y 312.513,Z 299.181,A -85,B 0,C 180,E1 -15693.689,E2 -15693.689} C_VEL
LIN {X 0,Y 312.513,Z 299.176,A -85,B 0,C 180,E1 -15697.387,E2 -15697.387} C_VEL
LIN {X 0,Y 312.485,Z 299.182,A -85,B 0,C 180,E1 -15700.71,E2 -15700.71} C_VEL
LIN {X 0,Y 312.447,Z 299.189,A -85,B 0,C 180,E1 -15704.211,E2 -15704.211} C_VEL
LIN {X 0,Y 312.48,Z 299.188,A -85,B 0,C 180,E1 -15707.92,E2 -15707.92} C_VEL
LIN {X 0,Y 312.487,Z 299.226,A -85,B 0,C 180,E1 -15711.632,E2 -15711.632} C_VEL
LIN {X 0,Y 312.911,Z 300.76,A -85,B 0,C 180,E1 -15712.088,E2 -15712.088} C_VEL
LIN {X 0,Y 320.588,Z 314.062,A -85,B 0,C 180,E1 -15713.522,E2 -15713.522} C_VEL
LIN {X 0,Y 329.376,Z 330.895,A -85,B 0,C 180,E1 -15715.095,E2 -15715.095} C_VEL
LIN {X 0,Y 337.809,Z 349.224,A -85,B 0,C 180,E1 -15716.555,E2 -15716.555} C_VEL
LIN {X 0,Y 334.783,Z 441.655,A -85,B 0,C 180,E1 -15718.522,E2 -15718.522} C_VEL
LIN {X 0,Y 333.784,Z 466.279,A -85,B 0,C 180,E1 -15719.078,E2 -15719.078} C_VEL
LIN {X 0,Y 332.751,Z 481.26,A -85,B 0,C 180,E1 -15719.64,E2 -15719.64} C_VEL
LIN {X 0,Y 331.262,Z 496.198,A -85,B 0,C 180,E1 -15720.441,E2 -15720.441} C_VEL
LIN {X 0,Y 329.766,Z 508.904,A -85,B 0,C 180,E1 -15721.347,E2 -15721.347} C_VEL
LIN {X 0,Y 327.634,Z 522.469,A -85,B 0,C 180,E1 -15722.537,E2 -15722.537} C_VEL
LIN {X 0,Y 325.513,Z 534.941,A -85,B 0,C 180,E1 -15723.903,E2 -15723.903} C_VEL
LIN {X 0,Y 323.211,Z 546.515,A -85,B 0,C 180,E1 -15725.427,E2 -15725.427} C_VEL
LIN {X 0,Y 321.108,Z 557.256,A -85,B 0,C 180,E1 -15727.14,E2 -15727.14} C_VEL
LIN {X 0,Y 318.907,Z 567.189,A -85,B 0,C 180,E1 -15729.016,E2 -15729.016} C_VEL
LIN {X 0,Y 316.775,Z 576.884,A -85,B 0,C 180,E1 -15731.235,E2 -15731.235} C_VEL
LIN {X 0,Y 314.919,Z 584.998,A -85,B 0,C 180,E1 -15733.481,E2 -15733.481} C_VEL
LIN {X 0,Y 313.62,Z 591.621,A -85,B 0,C 180,E1 -15735.73,E2 -15735.73} C_VEL
LIN {X 0,Y 312.373,Z 597.787,A -85,B 0,C 180,E1 -15738.318,E2 -15738.318} C_VEL
LIN {X 0,Y 311.596,Z 602.543,A -85,B 0,C 180,E1 -15740.916,E2 -15740.916} C_VEL
LIN {X 0,Y 311.057,Z 606.331,A -85,B 0,C 180,E1 -15743.791,E2 -15743.791} C_VEL
LIN {X 0,Y 310.875,Z 608.325,A -85,B 0,C 180,E1 -15746.111,E2 -15746.111} C_VEL
LIN {X 0,Y 310.692,Z 609.5,A -85,B 0,C 180,E1 -15748.704,E2 -15748.704} C_VEL
LIN {X 0,Y 310.692,Z 609.515,A -85,B 0,C 180,E1 -15751.296,E2 -15751.296} C_VEL
LIN {X 0,Y 310.869,Z 608.395,A -85,B 0,C 180,E1 -15753.889,E2 -15753.889} C_VEL
LIN {X 0,Y 311.104,Z 606.15,A -85,B 0,C 180,E1 -15756.485,E2 -15756.485} C_VEL
LIN {X 0,Y 311.573,Z 602.718,A -85,B 0,C 180,E1 -15759.085,E2 -15759.085} C_VEL
LIN {X 0,Y 312.34,Z 598.019,A -85,B 0,C 180,E1 -15761.683,E2 -15761.683} C_VEL
LIN {X 0,Y 313.589,Z 591.924,A -85,B 0,C 180,E1 -15764.272,E2 -15764.272} C_VEL
LIN {X 0,Y 315.129,Z 584.249,A -85,B 0,C 180,E1 -15766.853,E2 -15766.853} C_VEL
LIN {X 0,Y 316.966,Z 576.06,A -85,B 0,C 180,E1 -15769.089,E2 -15769.089} C_VEL
LIN {X 0,Y 319.148,Z 566.191,A -85,B 0,C 180,E1 -15771.305,E2 -15771.305} C_VEL
LIN {X 0,Y 321.383,Z 555.451,A -85,B 0,C 180,E1 -15773.298,E2 -15773.298} C_VEL
LIN {X 0,Y 323.789,Z 544.013,A -85,B 0,C 180,E1 -15775.04,E2 -15775.04} C_VEL
LIN {X 0,Y 326.064,Z 531.919,A -85,B 0,C 180,E1 -15776.566,E2 -15776.566} C_VEL
LIN {X 0,Y 328.33,Z 518.771,A -85,B 0,C 180,E1 -15777.919,E2 -15777.919} C_VEL
LIN {X 0,Y 330.244,Z 505.455,A -85,B 0,C 180,E1 -15779.025,E2 -15779.025} C_VEL
LIN {X 0,Y 331.801,Z 491.575,A -85,B 0,C 180,E1 -15779.938,E2 -15779.938} C_VEL
LIN {X 0,Y 333.176,Z 476.301,A -85,B 0,C 180,E1 -15780.677,E2 -15780.677} C_VEL
LIN {X 0,Y 334.166,Z 461.572,A -85,B 0,C 180,E1 -15781.146,E2 -15781.146} C_VEL
LIN {X 0,Y 336.331,Z 398.411,A -85,B 0,C 180,E1 -15782.498,E2 -15782.498} C_VEL
LIN {X 0,Y 335.978,Z 392.614,A -85,B 0,C 180,E1 -15782.681,E2 -15782.681} C_VEL
LIN {X 0,Y 331.794,Z 374.011,A -85,B 0,C 180,E1 -15783.622,E2 -15783.622} C_VEL
LIN {X 0,Y 331.406,Z 368.216,A -85,B 0,C 180,E1 -15783.815,E2 -15783.815} C_VEL
LIN {X 0,Y 331.922,Z 351.428,A -85,B 0,C 180,E1 -15784.185,E2 -15784.185} C_VEL
LIN {X 0,Y 323.722,Z 333.58,A -85,B 0,C 180,E1 -15785.66,E2 -15785.66} C_VEL
LIN {X 0,Y 314.648,Z 316.273,A -85,B 0,C 180,E1 -15787.349,E2 -15787.349} C_VEL
LIN {X 0,Y 307.651,Z 304.389,A -85,B 0,C 180,E1 -15788.705,E2 -15788.705} C_VEL
LIN {X 0,Y 305.872,Z 301.733,A -85,B 0,C 180,E1 -15789.053,E2 -15789.053} C_VEL
LIN {X 0,Y 305.544,Z 300.6,A -85,B 0,C 180,E1 -15789.189,E2 -15789.189} C_VEL
LIN {X 0,Y 305.467,Z 300.057,A -85,B 0,C 180,E1 -15789.383,E2 -15789.383} C_VEL
LIN {X 0,Y 305.451,Z 300.063,A -85,B 0,C 180,E1 -15792.585,E2 -15792.585} C_VEL
LIN {X 0,Y 305.421,Z 300.066,A -85,B 0,C 180,E1 -15796.344,E2 -15796.344} C_VEL
LIN {X 0,Y 305.453,Z 300.058,A -85,B 0,C 180,E1 -15799.891,E2 -15799.891} C_VEL
LIN {X 0,Y 305.458,Z 300.039,A -85,B 0,C 180,E1 -15803.635,E2 -15803.635} C_VEL
LIN {X 0,Y 305.459,Z 300.061,A -85,B 0,C 180,E1 -15806.482,E2 -15806.482} C_VEL
LIN {X 0,Y 305.429,Z 300.036,A -85,B 0,C 180,E1 -15809.587,E2 -15809.587} C_VEL
LIN {X 0,Y 305.477,Z 300.059,A -85,B 0,C 180,E1 -15812.604,E2 -15812.604} C_VEL
LIN {X 0,Y 305.483,Z 300.057,A -85,B 0,C 180,E1 -15815.536,E2 -15815.536} C_VEL
LIN {X 0,Y 305.488,Z 300.056,A -85,B 0,C 180,E1 -15819.813,E2 -15819.813} C_VEL
LIN {X 0,Y 305.533,Z 300.043,A -85,B 0,C 180,E1 -15822.6,E2 -15822.6} C_VEL
LIN {X 0,Y 305.618,Z 300.037,A -85,B 0,C 180,E1 -15825.347,E2 -15825.347} C_VEL
LIN {X 0,Y 305.615,Z 300.039,A -85,B 0,C 180,E1 -15829.399,E2 -15829.399} C_VEL
